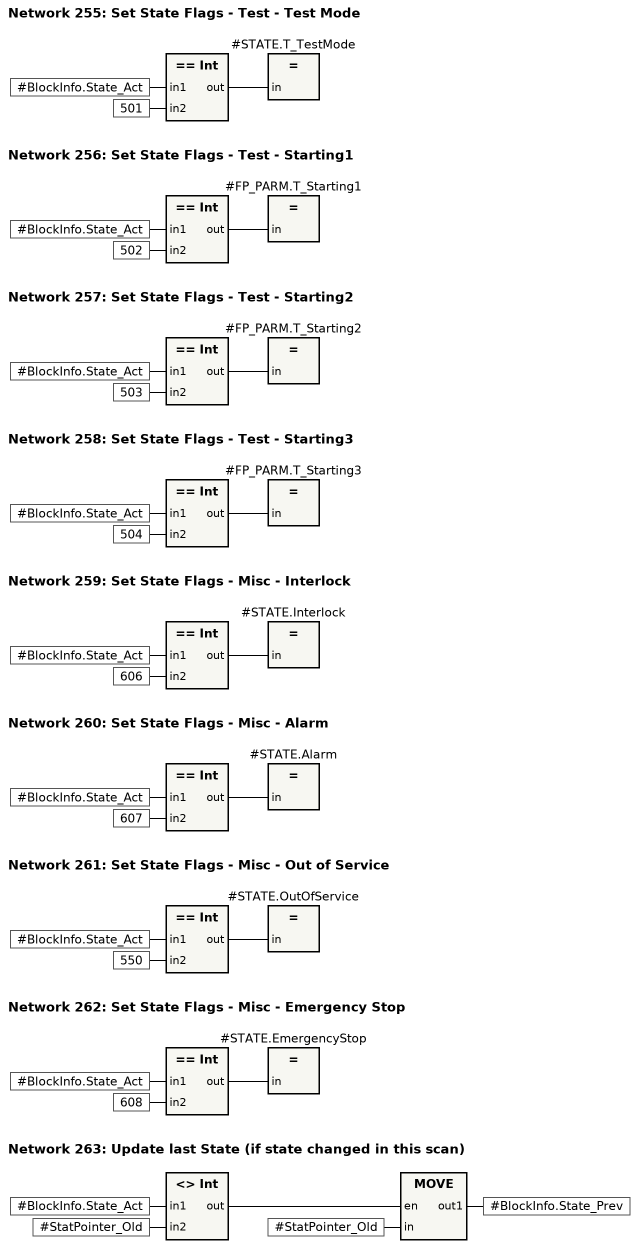
   #STATE.T_TestMode := #BlockInfo.State_Act = 501;
END_REGION

REGION Network 256: Set State Flags - Test - Starting1
   #FP_PARM.T_Starting1 := #BlockInfo.State_Act = 502;
END_REGION

REGION Network 257: Set State Flags - Test - Starting2
   #FP_PARM.T_Starting2 := #BlockInfo.State_Act = 503;
END_REGION

REGION Network 258: Set State Flags - Test - Starting3
   #FP_PARM.T_Starting3 := #BlockInfo.State_Act = 504;
END_REGION

REGION Network 259: Set State Flags - Misc - Interlock
   #STATE.Interlock := #BlockInfo.State_Act = 606;
END_REGION

REGION Network 260: Set State Flags - Misc - Alarm
   #STATE.Alarm := #BlockInfo.State_Act = 607;
END_REGION

REGION Network 261: Set State Flags - Misc - Out of Service
   #STATE.OutOfService := #BlockInfo.State_Act = 550;
END_REGION

REGION Network 262: Set State Flags - Misc - Emergency Stop
   #STATE.EmergencyStop := #BlockInfo.State_Act = 608;
END_REGION

REGION Network 263: Update last State (if state changed in this scan)
   IF #BlockInfo.State_Act <> #StatPointer_Old THEN #BlockInfo.State_Prev := #StatPointer_Old; END_IF;
END_REGION

REGION Network 264: Update MSW
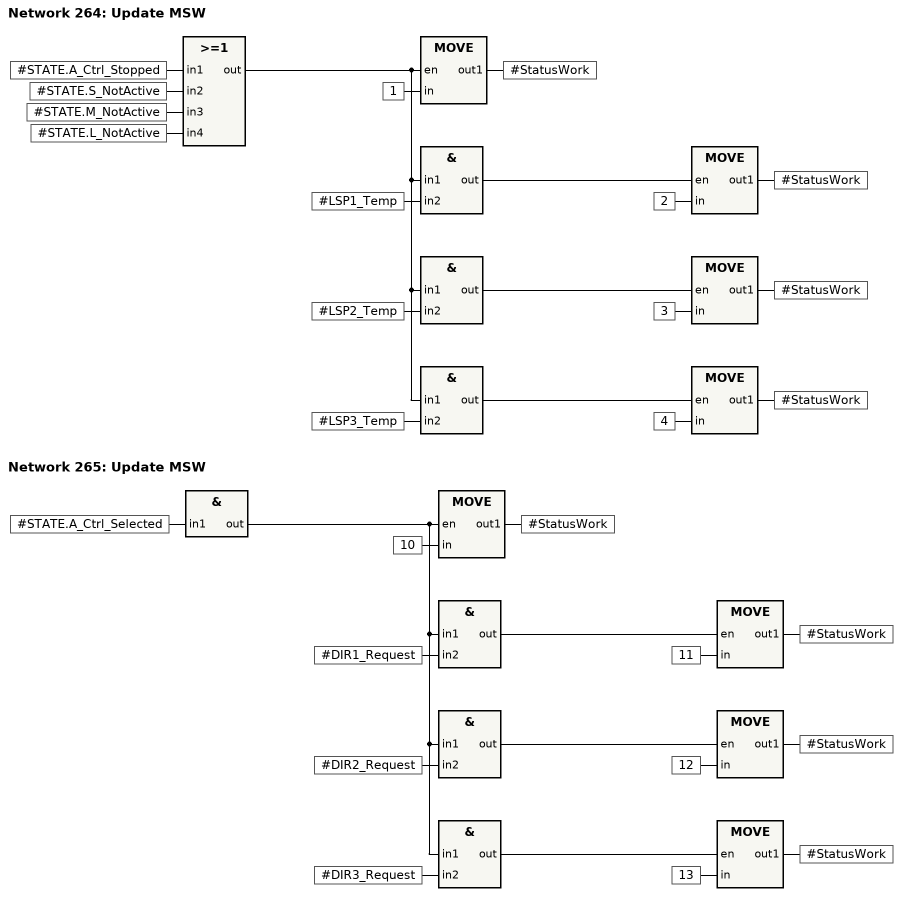
   #_w1 := #STATE.A_Ctrl_Stopped OR #STATE.S_NotActive OR #STATE.M_NotActive OR #STATE.L_NotActive;
   IF #_w1 THEN #StatusWork := 1; END_IF;
   IF #_w1 AND #LSP1_Temp THEN #StatusWork := 2; END_IF;
   IF #_w1 AND #LSP2_Temp THEN #StatusWork := 3; END_IF;
   IF #_w1 AND #LSP3_Temp THEN #StatusWork := 4; END_IF;
END_REGION

REGION Network 265: Update MSW
   IF #STATE.A_Ctrl_Selected THEN #StatusWork := 10; END_IF;
   IF #STATE.A_Ctrl_Selected AND #DIR1_Request THEN #StatusWork := 11; END_IF;
   IF #STATE.A_Ctrl_Selected AND #DIR2_Request THEN #StatusWork := 12; END_IF;
   IF #STATE.A_Ctrl_Selected AND #DIR3_Request THEN #StatusWork := 13; END_IF;
END_REGION

REGION Network 266: Update MSW
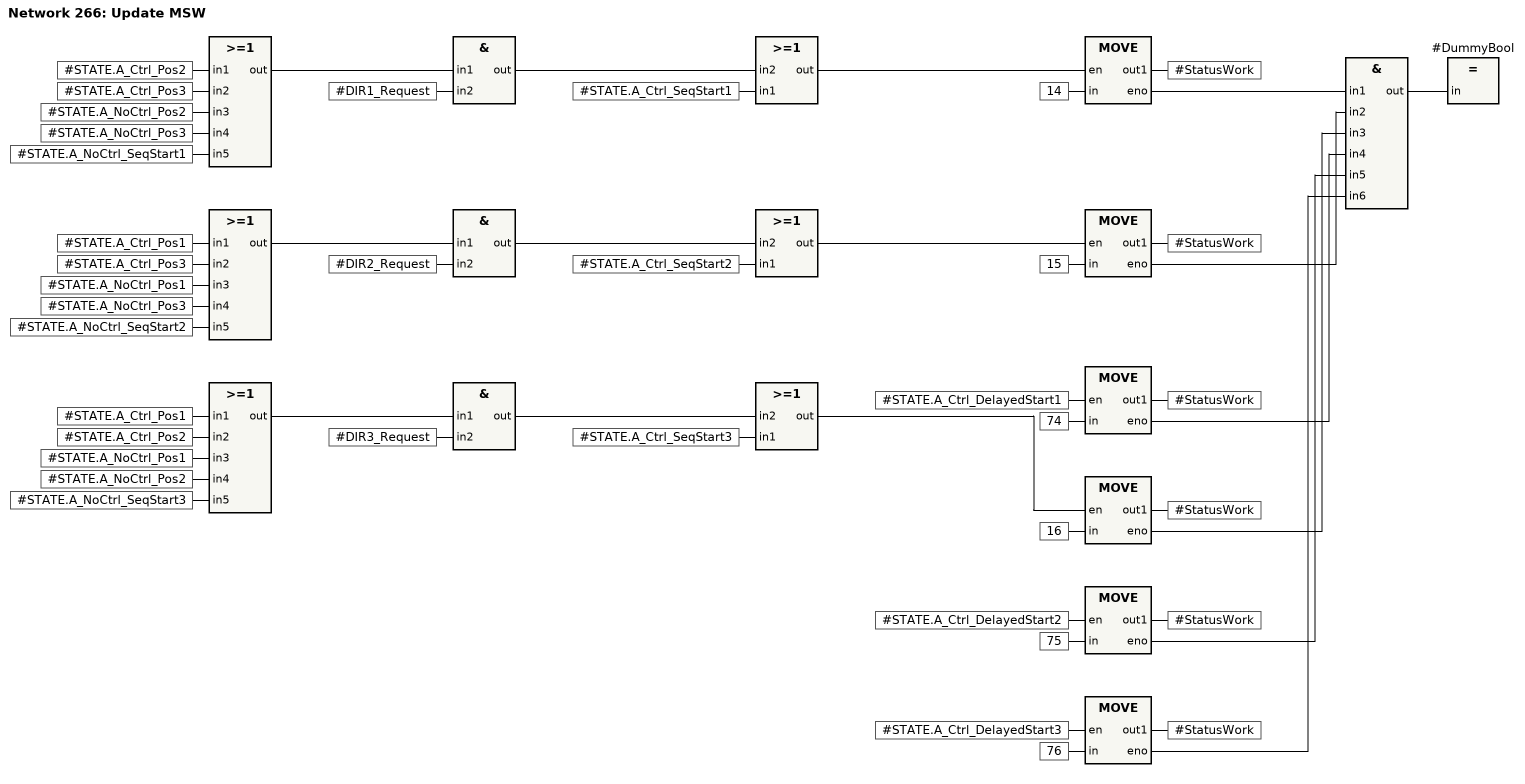
   // ENO of a box is taken as its EN; it also drops when the box reports an error
   #_w1 := ((#STATE.A_Ctrl_Pos2 OR #STATE.A_Ctrl_Pos3 OR #STATE.A_NoCtrl_Pos2 OR #STATE.A_NoCtrl_Pos3 OR #STATE.A_NoCtrl_SeqStart1) AND #DIR1_Request) OR #STATE.A_Ctrl_SeqStart1;
   IF #_w1 THEN #StatusWork := 14; END_IF;
   #_w2 := ((#STATE.A_Ctrl_Pos1 OR #STATE.A_Ctrl_Pos3 OR #STATE.A_NoCtrl_Pos1 OR #STATE.A_NoCtrl_Pos3 OR #STATE.A_NoCtrl_SeqStart2) AND #DIR2_Request) OR #STATE.A_Ctrl_SeqStart2;
   IF #_w2 THEN #StatusWork := 15; END_IF;
   #_w3 := ((#STATE.A_Ctrl_Pos1 OR #STATE.A_Ctrl_Pos2 OR #STATE.A_NoCtrl_Pos1 OR #STATE.A_NoCtrl_Pos2 OR #STATE.A_NoCtrl_SeqStart3) AND #DIR3_Request) OR #STATE.A_Ctrl_SeqStart3;
   IF #_w3 THEN #StatusWork := 16; END_IF;
   IF #STATE.A_Ctrl_DelayedStart1 THEN #StatusWork := 74; END_IF;
   IF #STATE.A_Ctrl_DelayedStart2 THEN #StatusWork := 75; END_IF;
   IF #STATE.A_Ctrl_DelayedStart3 THEN #StatusWork := 76; END_IF;
   #DummyBool := #_w1 AND #_w2 AND #_w3 AND #STATE.A_Ctrl_DelayedStart1 AND #STATE.A_Ctrl_DelayedStart2 AND #STATE.A_Ctrl_DelayedStart3;
END_REGION

REGION Network 267: Update MSW
   // Build 007 - 30.09.2020 (EXTBOB):  State Alarm Neg added to avoid start warn in case of alarm state
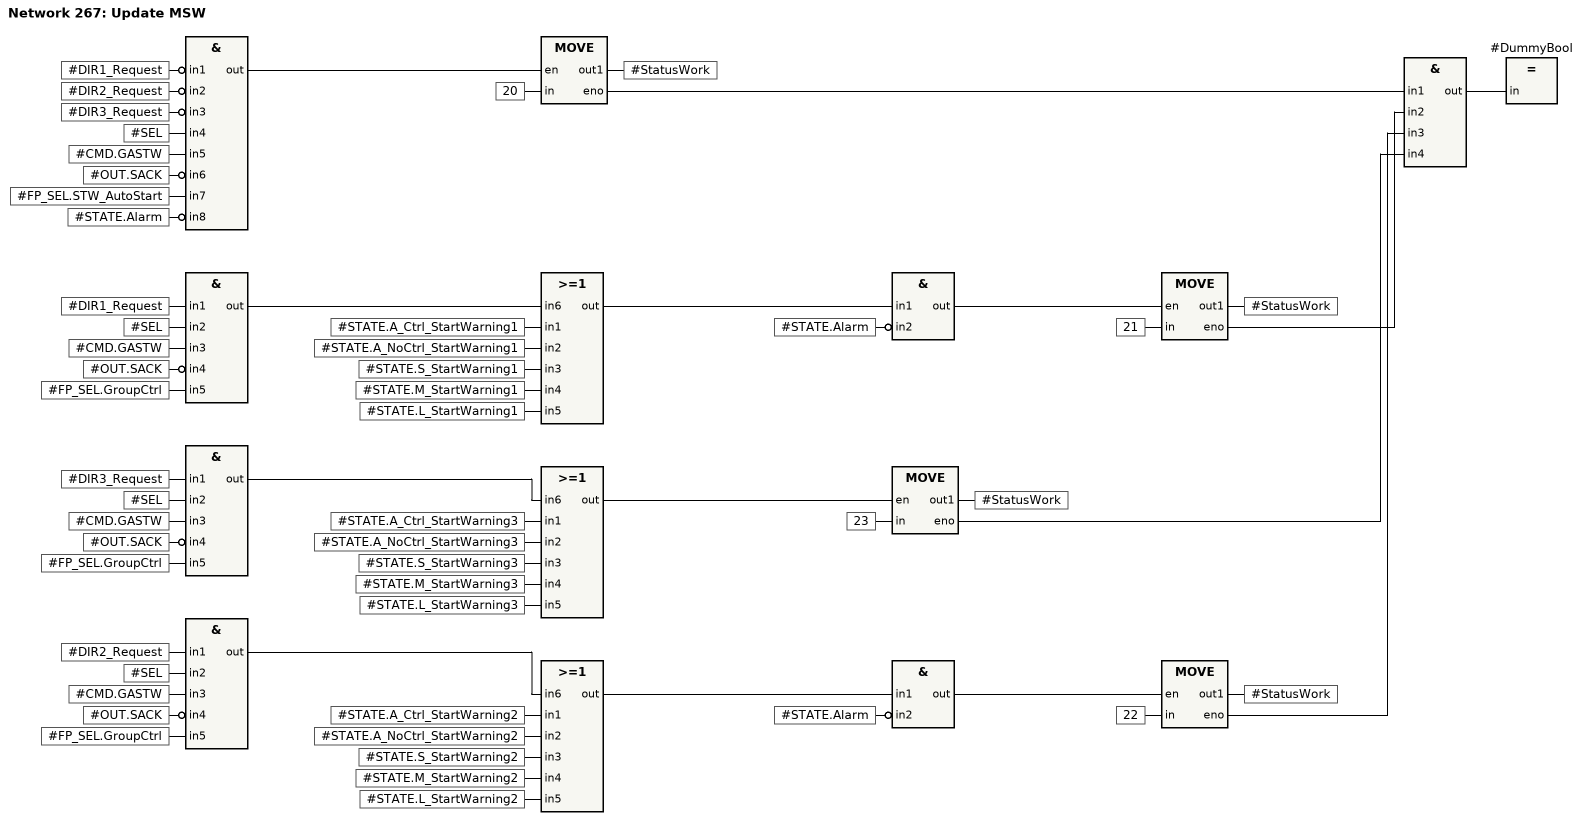
   // ENO of a box is taken as its EN; it also drops when the box reports an error
   #_w1 := NOT #DIR1_Request AND NOT #DIR2_Request AND NOT #DIR3_Request AND #SEL AND #CMD.GASTW AND NOT #OUT.SACK AND #FP_SEL.STW_AutoStart AND NOT #STATE.Alarm;
   IF #_w1 THEN #StatusWork := 20; END_IF;
   #_w2 := ((#DIR1_Request AND #SEL AND #CMD.GASTW AND NOT #OUT.SACK AND #FP_SEL.GroupCtrl) OR #STATE.A_Ctrl_StartWarning1 OR #STATE.A_NoCtrl_StartWarning1 OR #STATE.S_StartWarning1 OR #STATE.M_StartWarning1 OR #STATE.L_StartWarning1) AND NOT #STATE.Alarm;
   IF #_w2 THEN #StatusWork := 21; END_IF;
   #_w3 := ((#DIR2_Request AND #SEL AND #CMD.GASTW AND NOT #OUT.SACK AND #FP_SEL.GroupCtrl) OR #STATE.A_Ctrl_StartWarning2 OR #STATE.A_NoCtrl_StartWarning2 OR #STATE.S_StartWarning2 OR #STATE.M_StartWarning2 OR #STATE.L_StartWarning2) AND NOT #STATE.Alarm;
   IF #_w3 THEN #StatusWork := 22; END_IF;
   #_w4 := (#DIR3_Request AND #SEL AND #CMD.GASTW AND NOT #OUT.SACK AND #FP_SEL.GroupCtrl) OR #STATE.A_Ctrl_StartWarning3 OR #STATE.A_NoCtrl_StartWarning3 OR #STATE.S_StartWarning3 OR #STATE.M_StartWarning3 OR #STATE.L_StartWarning3;
   IF #_w4 THEN #StatusWork := 23; END_IF;
   #DummyBool := #_w1 AND #_w2 AND #_w3 AND #_w4;
END_REGION

REGION Network 268: Update MSW
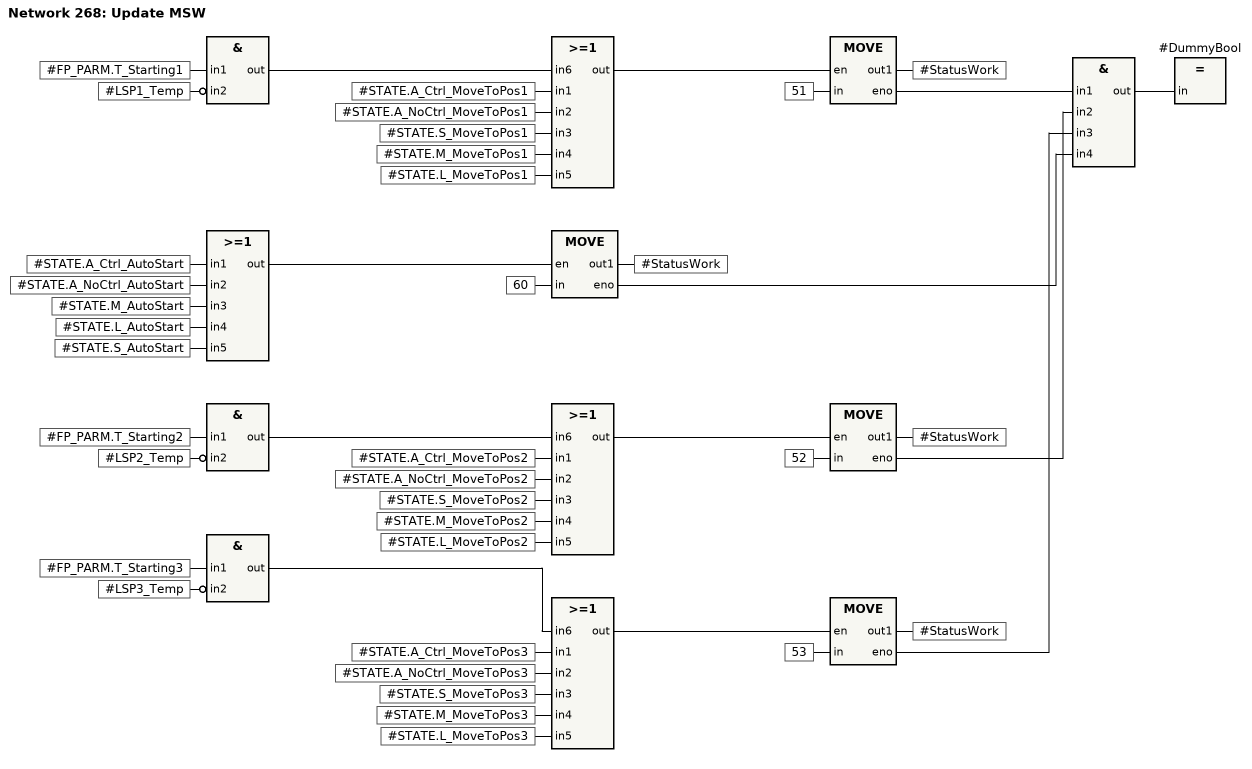
   // ENO of a box is taken as its EN; it also drops when the box reports an error
   #_w1 := (#FP_PARM.T_Starting1 AND NOT #LSP1_Temp) OR #STATE.A_Ctrl_MoveToPos1 OR #STATE.A_NoCtrl_MoveToPos1 OR #STATE.S_MoveToPos1 OR #STATE.M_MoveToPos1 OR #STATE.L_MoveToPos1;
   IF #_w1 THEN #StatusWork := 51; END_IF;
   #_w2 := (#FP_PARM.T_Starting2 AND NOT #LSP2_Temp) OR #STATE.A_Ctrl_MoveToPos2 OR #STATE.A_NoCtrl_MoveToPos2 OR #STATE.S_MoveToPos2 OR #STATE.M_MoveToPos2 OR #STATE.L_MoveToPos2;
   IF #_w2 THEN #StatusWork := 52; END_IF;
   #_w3 := (#FP_PARM.T_Starting3 AND NOT #LSP3_Temp) OR #STATE.A_Ctrl_MoveToPos3 OR #STATE.A_NoCtrl_MoveToPos3 OR #STATE.S_MoveToPos3 OR #STATE.M_MoveToPos3 OR #STATE.L_MoveToPos3;
   IF #_w3 THEN #StatusWork := 53; END_IF;
   #_w4 := #STATE.A_Ctrl_AutoStart OR #STATE.A_NoCtrl_AutoStart OR #STATE.M_AutoStart OR #STATE.L_AutoStart OR #STATE.S_AutoStart;
   IF #_w4 THEN #StatusWork := 60; END_IF;
   #DummyBool := #_w1 AND #_w2 AND #_w3 AND #_w4;
END_REGION

REGION Network 269: Update MSW
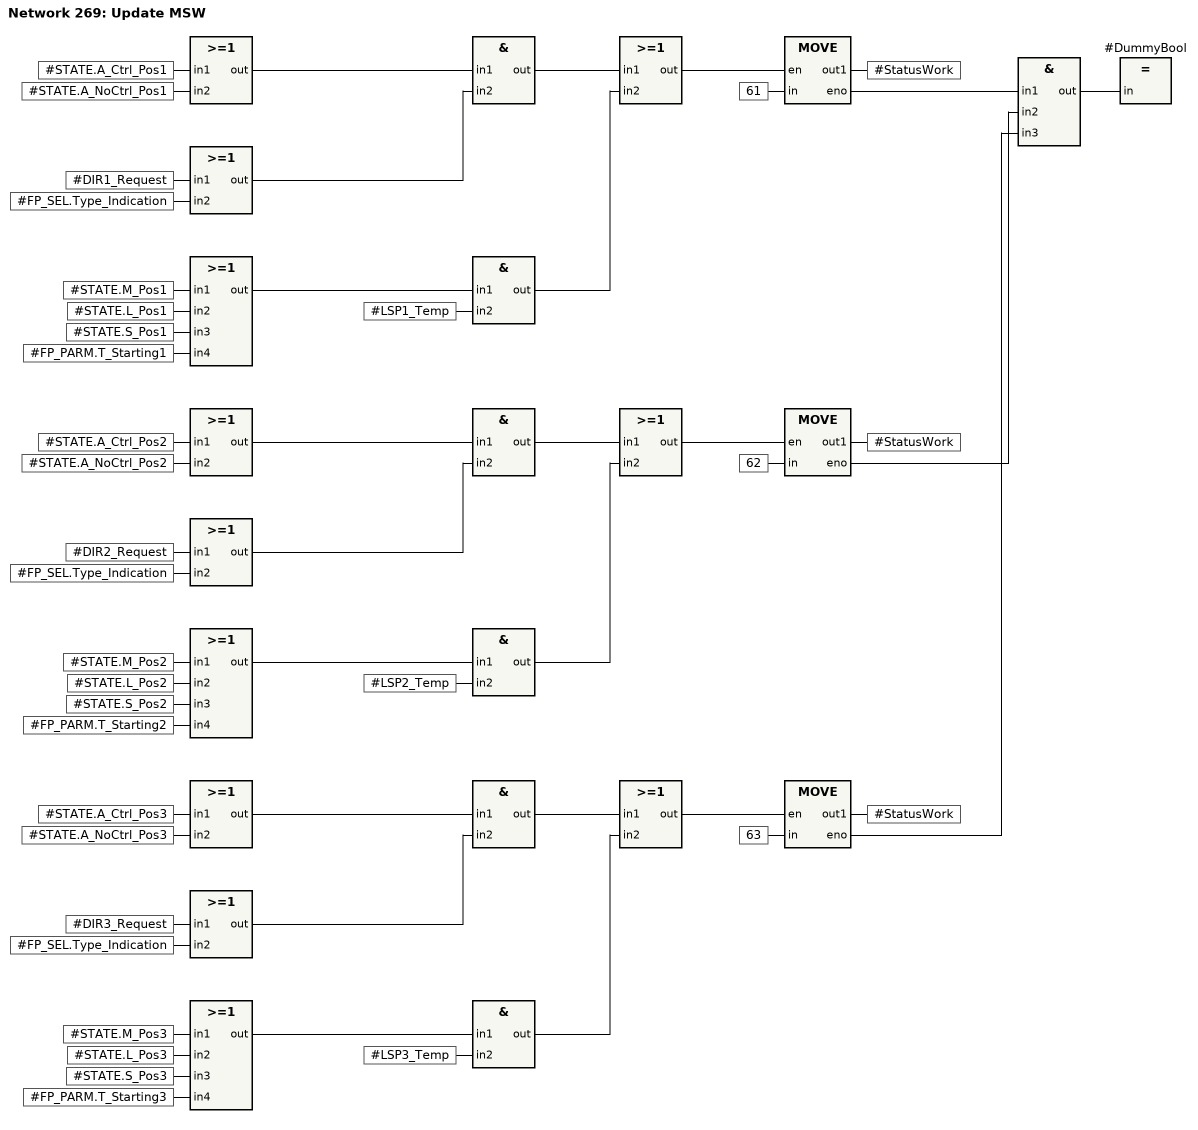
   // ENO of a box is taken as its EN; it also drops when the box reports an error
   #_w1 := ((#STATE.A_Ctrl_Pos1 OR #STATE.A_NoCtrl_Pos1) AND (#DIR1_Request OR #FP_SEL.Type_Indication)) OR ((#STATE.M_Pos1 OR #STATE.L_Pos1 OR #STATE.S_Pos1 OR #FP_PARM.T_Starting1) AND #LSP1_Temp);
   IF #_w1 THEN #StatusWork := 61; END_IF;
   #_w2 := ((#STATE.A_Ctrl_Pos2 OR #STATE.A_NoCtrl_Pos2) AND (#DIR2_Request OR #FP_SEL.Type_Indication)) OR ((#STATE.M_Pos2 OR #STATE.L_Pos2 OR #STATE.S_Pos2 OR #FP_PARM.T_Starting2) AND #LSP2_Temp);
   IF #_w2 THEN #StatusWork := 62; END_IF;
   #_w3 := ((#STATE.A_Ctrl_Pos3 OR #STATE.A_NoCtrl_Pos3) AND (#DIR3_Request OR #FP_SEL.Type_Indication)) OR ((#STATE.M_Pos3 OR #STATE.L_Pos3 OR #STATE.S_Pos3 OR #FP_PARM.T_Starting3) AND #LSP3_Temp);
   IF #_w3 THEN #StatusWork := 63; END_IF;
   #DummyBool := #_w1 AND #_w2 AND #_w3;
END_REGION

REGION Network 270: Update MSW
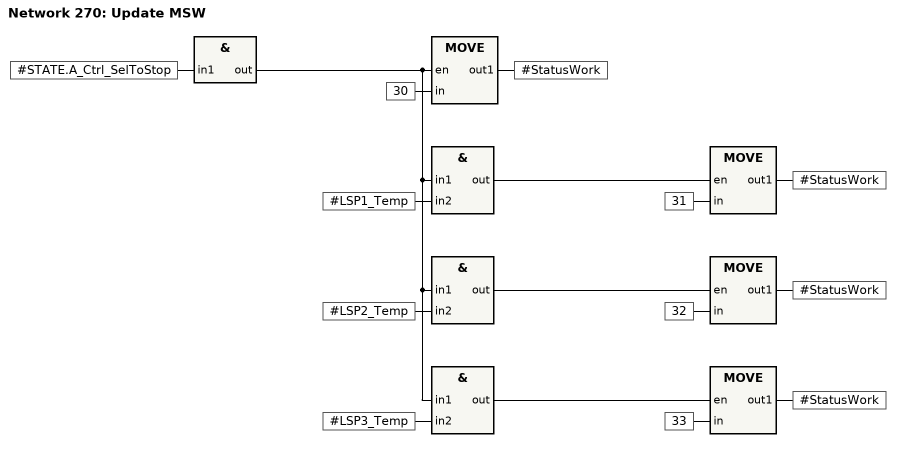
   IF #STATE.A_Ctrl_SelToStop THEN #StatusWork := 30; END_IF;
   IF #STATE.A_Ctrl_SelToStop AND #LSP1_Temp THEN #StatusWork := 31; END_IF;
   IF #STATE.A_Ctrl_SelToStop AND #LSP2_Temp THEN #StatusWork := 32; END_IF;
   IF #STATE.A_Ctrl_SelToStop AND #LSP3_Temp THEN #StatusWork := 33; END_IF;
END_REGION

REGION Network 271: Update MSW
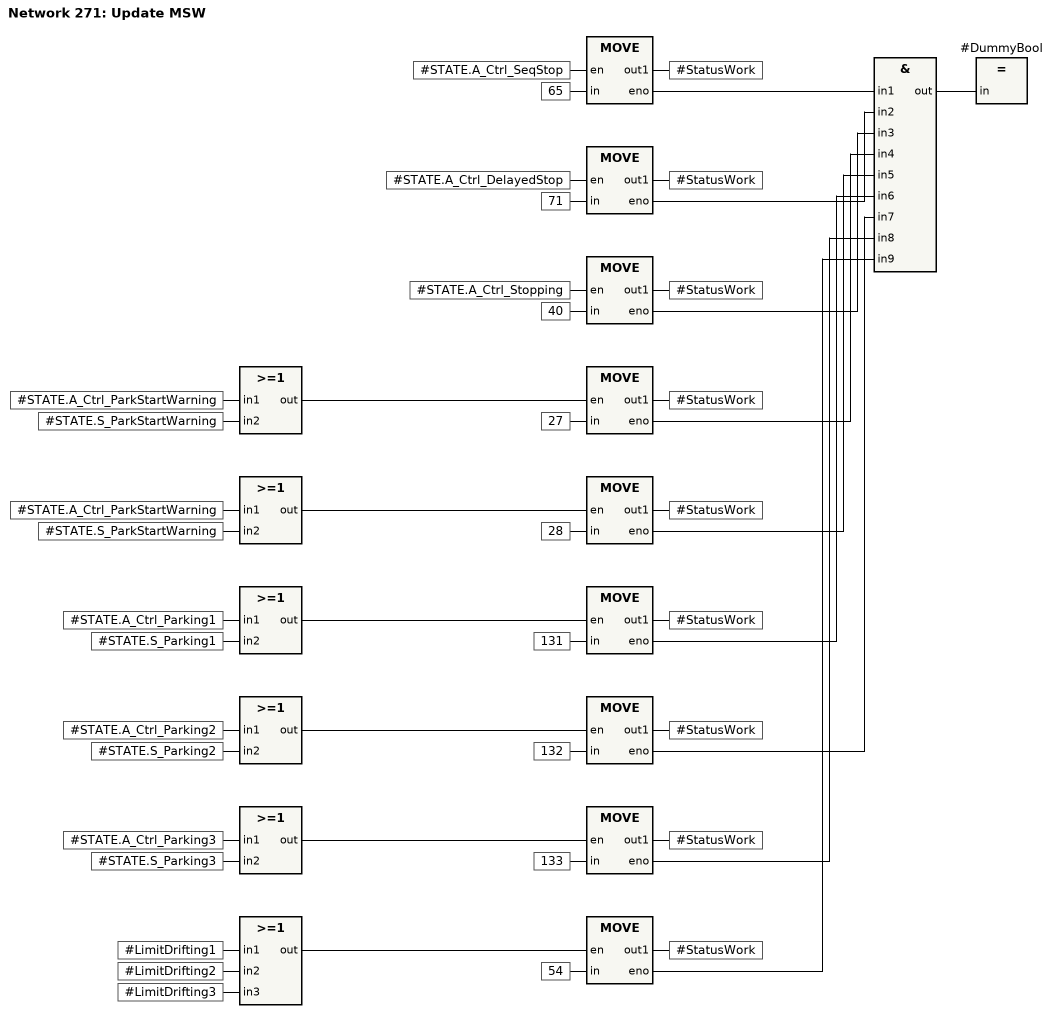
   // ENO of a box is taken as its EN; it also drops when the box reports an error
   IF #STATE.A_Ctrl_SeqStop THEN #StatusWork := 65; END_IF;
   IF #STATE.A_Ctrl_DelayedStop THEN #StatusWork := 71; END_IF;
   IF #STATE.A_Ctrl_Stopping THEN #StatusWork := 40; END_IF;
   #_w1 := #STATE.A_Ctrl_ParkStartWarning OR #STATE.S_ParkStartWarning;
   IF #_w1 THEN #StatusWork := 27; END_IF;
   #_w2 := #STATE.A_Ctrl_ParkStartWarning OR #STATE.S_ParkStartWarning;
   IF #_w2 THEN #StatusWork := 28; END_IF;
   #_w3 := #STATE.A_Ctrl_Parking1 OR #STATE.S_Parking1;
   IF #_w3 THEN #StatusWork := 131; END_IF;
   #_w4 := #STATE.A_Ctrl_Parking2 OR #STATE.S_Parking2;
   IF #_w4 THEN #StatusWork := 132; END_IF;
   #_w5 := #STATE.A_Ctrl_Parking3 OR #STATE.S_Parking3;
   IF #_w5 THEN #StatusWork := 133; END_IF;
   #_w6 := #LimitDrifting1 OR #LimitDrifting2 OR #LimitDrifting3;
   IF #_w6 THEN #StatusWork := 54; END_IF;
   #DummyBool := #STATE.A_Ctrl_SeqStop AND #STATE.A_Ctrl_DelayedStop AND #STATE.A_Ctrl_Stopping AND #_w1 AND #_w2 AND #_w3 AND #_w4 AND #_w5 AND #_w6;
END_REGION

REGION Network 272: Update MSW
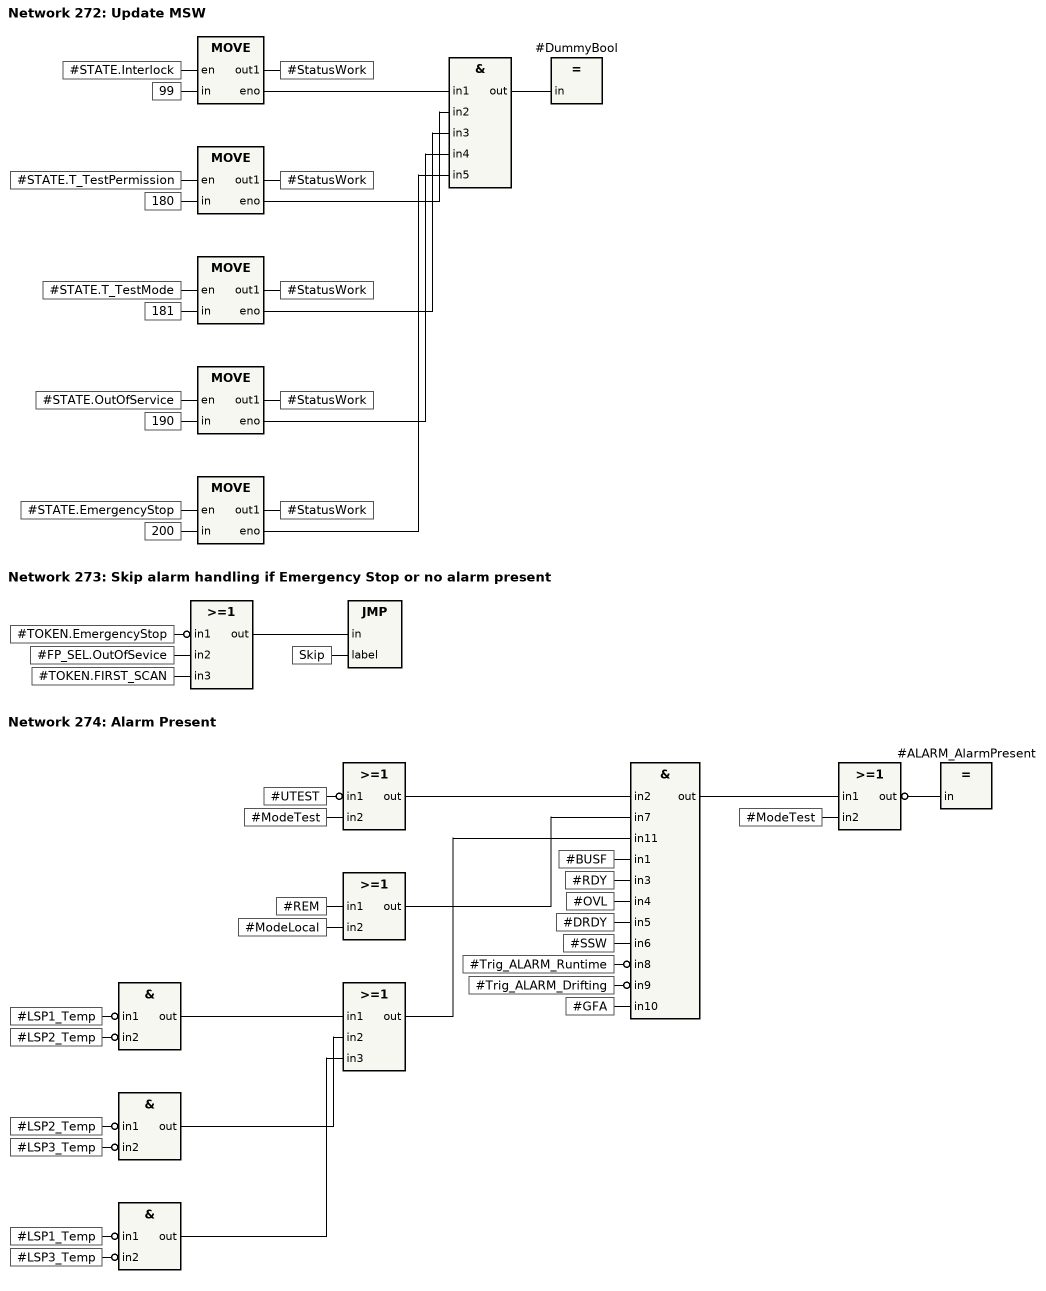
   // ENO of a box is taken as its EN; it also drops when the box reports an error
   IF #STATE.Interlock THEN #StatusWork := 99; END_IF;
   IF #STATE.T_TestPermission THEN #StatusWork := 180; END_IF;
   IF #STATE.T_TestMode THEN #StatusWork := 181; END_IF;
   IF #STATE.OutOfService THEN #StatusWork := 190; END_IF;
   IF #STATE.EmergencyStop THEN #StatusWork := 200; END_IF;
   #DummyBool := #STATE.Interlock AND #STATE.T_TestPermission AND #STATE.T_TestMode AND #STATE.OutOfService AND #STATE.EmergencyStop;
END_REGION

REGION Network 273: Skip alarm handling if Emergency Stop or no alarm present
   // Skip = Skip Alarm
   IF NOT #TOKEN.EmergencyStop OR #FP_SEL.OutOfSevice OR #TOKEN.FIRST_SCAN THEN GOTO Skip; END_IF;
END_REGION

REGION Network 274: Alarm Present
   #ALARM_AlarmPresent := NOT (((NOT #UTEST OR #ModeTest) AND (#REM OR #ModeLocal) AND ((NOT #LSP1_Temp AND NOT #LSP2_Temp) OR (NOT #LSP2_Temp AND NOT #LSP3_Temp) OR (NOT #LSP1_Temp AND NOT #LSP3_Temp)) AND #BUSF AND #RDY AND #OVL AND #DRDY AND #SSW AND NOT #Trig_ALARM_Runtime AND NOT #Trig_ALARM_Drifting AND #GFA) OR #ModeTest);
END_REGION

REGION Network 275: Alarm Warn Present
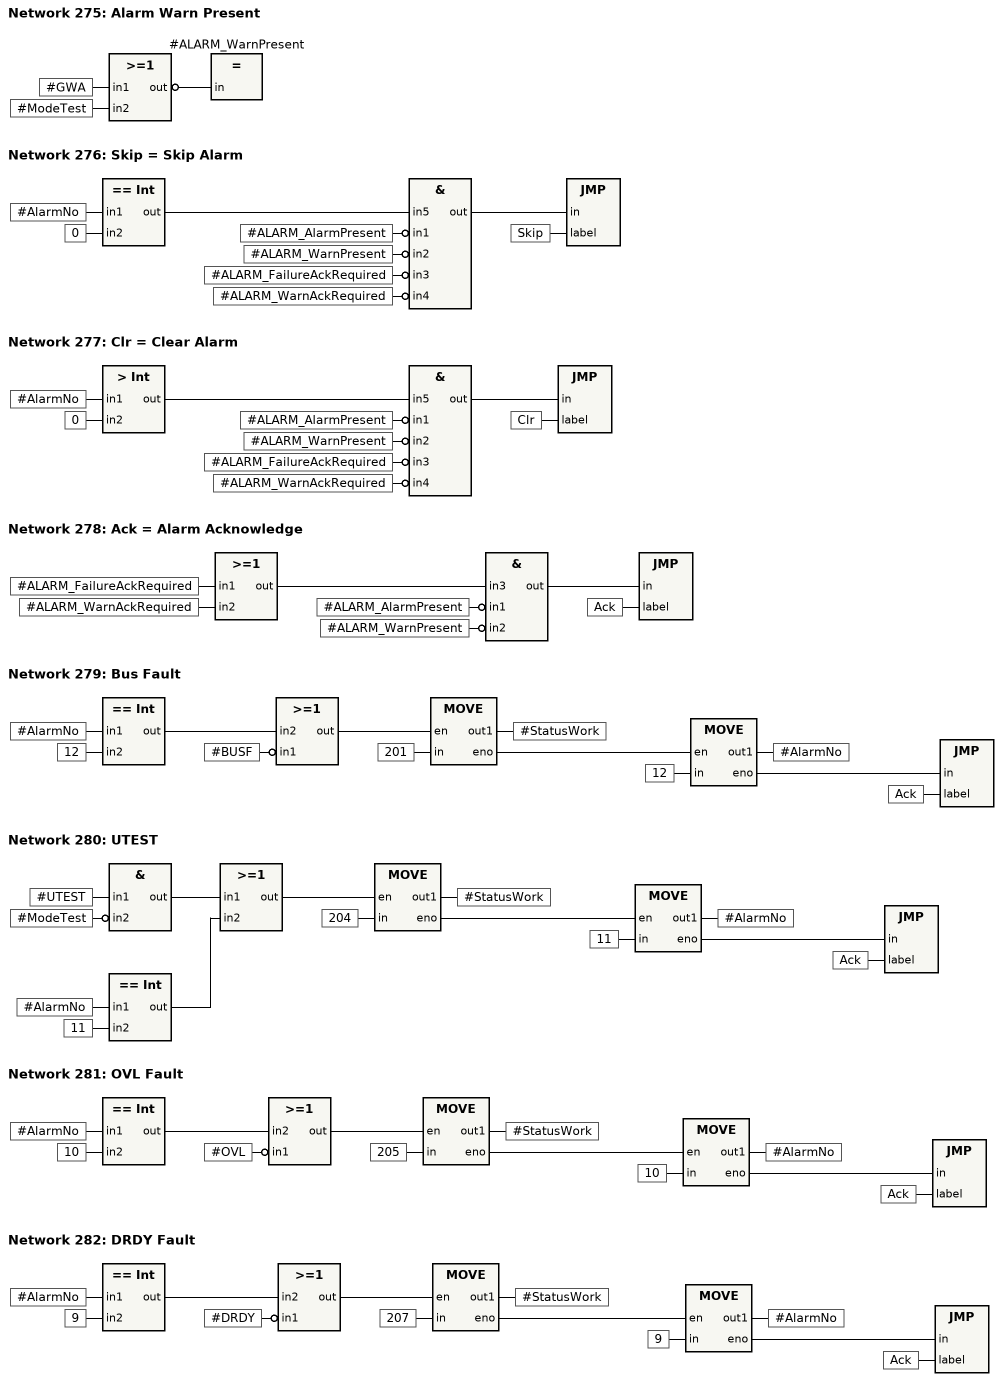
   #ALARM_WarnPresent := NOT (#GWA OR #ModeTest);
END_REGION

REGION Network 276: Skip = Skip Alarm
   IF (#AlarmNo = 0) AND NOT #ALARM_AlarmPresent AND NOT #ALARM_WarnPresent AND NOT #ALARM_FailureAckRequired AND NOT #ALARM_WarnAckRequired THEN
       GOTO Skip;
   END_IF;
END_REGION

REGION Network 277: Clr = Clear Alarm
   IF (#AlarmNo > 0) AND NOT #ALARM_AlarmPresent AND NOT #ALARM_WarnPresent AND NOT #ALARM_FailureAckRequired AND NOT #ALARM_WarnAckRequired THEN
       GOTO Clr;
   END_IF;
END_REGION

REGION Network 278: Ack = Alarm Acknowledge
   IF (#ALARM_FailureAckRequired OR #ALARM_WarnAckRequired) AND NOT #ALARM_AlarmPresent AND NOT #ALARM_WarnPresent THEN
       GOTO Ack;
   END_IF;
END_REGION

REGION Network 279: Bus Fault
   // ENO of a box is taken as its EN; it also drops when the box reports an error
   #_w1 := (#AlarmNo = 12) OR NOT #BUSF;
   IF #_w1 THEN
       #StatusWork := 201;
       #AlarmNo := 12;
       GOTO Ack;
   END_IF;
END_REGION

REGION Network 280: UTEST
   // ENO of a box is taken as its EN; it also drops when the box reports an error
   #_w1 := (#UTEST AND NOT #ModeTest) OR (#AlarmNo = 11);
   IF #_w1 THEN
       #StatusWork := 204;
       #AlarmNo := 11;
       GOTO Ack;
   END_IF;
END_REGION

REGION Network 281: OVL Fault
   // ENO of a box is taken as its EN; it also drops when the box reports an error
   #_w1 := (#AlarmNo = 10) OR NOT #OVL;
   IF #_w1 THEN
       #StatusWork := 205;
       #AlarmNo := 10;
       GOTO Ack;
   END_IF;
END_REGION

REGION Network 282: DRDY Fault
   // ENO of a box is taken as its EN; it also drops when the box reports an error
   #_w1 := (#AlarmNo = 9) OR NOT #DRDY;
   IF #_w1 THEN
       #StatusWork := 207;
       #AlarmNo := 9;
       GOTO Ack;
   END_IF;
END_REGION

REGION Network 283: RDY Fault
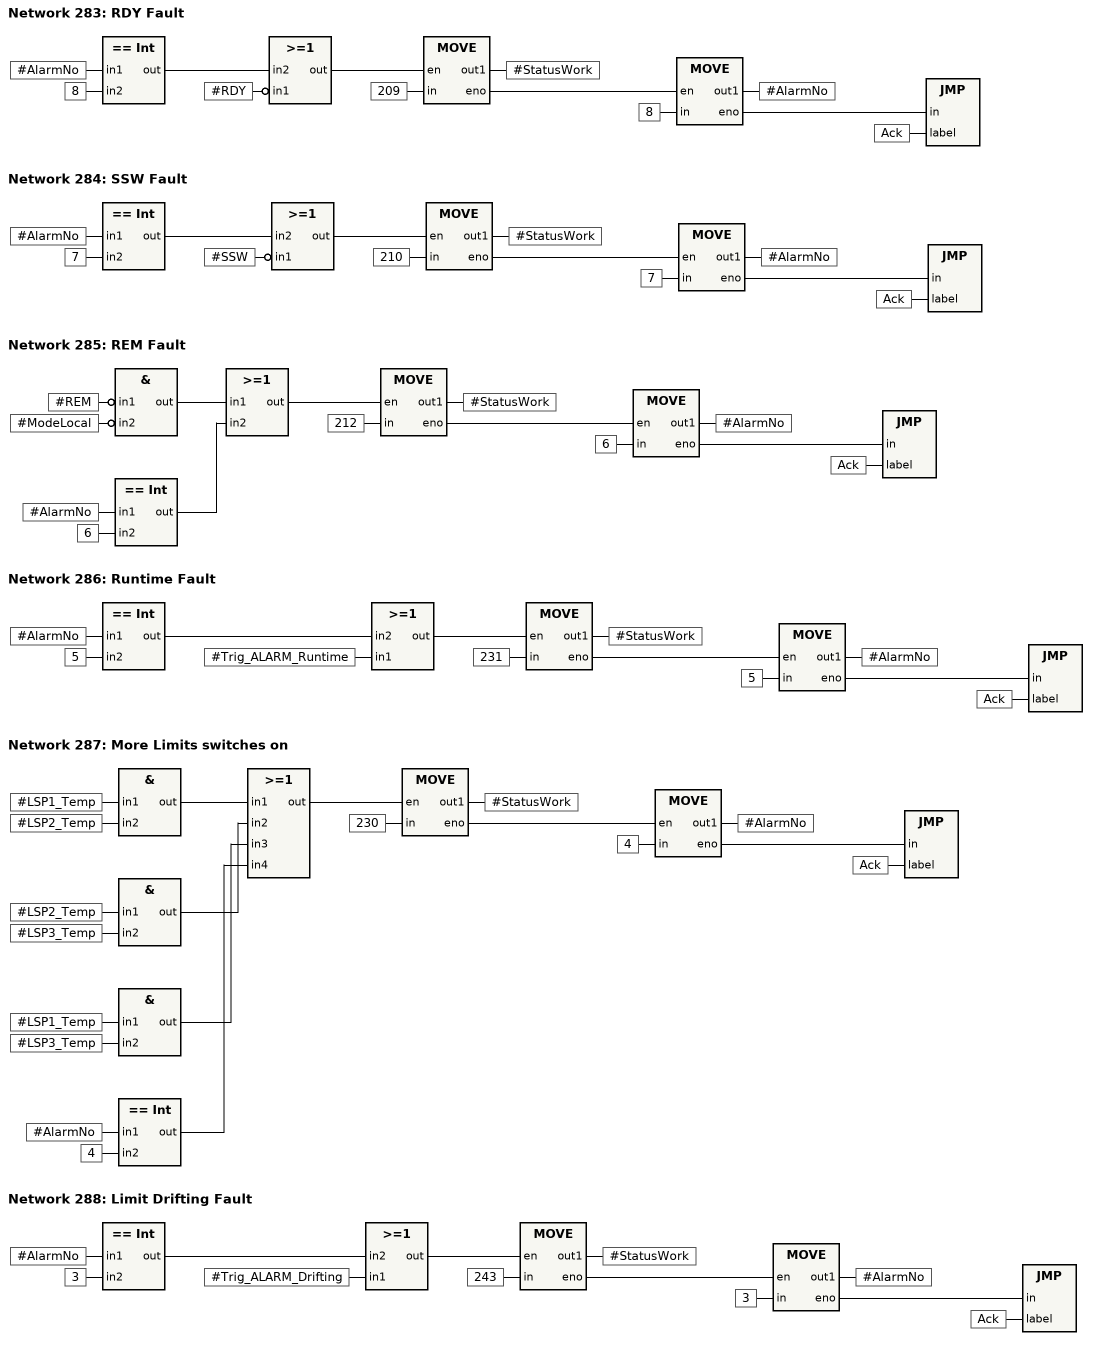
   // ENO of a box is taken as its EN; it also drops when the box reports an error
   #_w1 := (#AlarmNo = 8) OR NOT #RDY;
   IF #_w1 THEN
       #StatusWork := 209;
       #AlarmNo := 8;
       GOTO Ack;
   END_IF;
END_REGION

REGION Network 284: SSW Fault
   // ENO of a box is taken as its EN; it also drops when the box reports an error
   #_w1 := (#AlarmNo = 7) OR NOT #SSW;
   IF #_w1 THEN
       #StatusWork := 210;
       #AlarmNo := 7;
       GOTO Ack;
   END_IF;
END_REGION

REGION Network 285: REM Fault
   // ENO of a box is taken as its EN; it also drops when the box reports an error
   #_w1 := (NOT #REM AND NOT #ModeLocal) OR (#AlarmNo = 6);
   IF #_w1 THEN
       #StatusWork := 212;
       #AlarmNo := 6;
       GOTO Ack;
   END_IF;
END_REGION

REGION Network 286: Runtime Fault
   // ENO of a box is taken as its EN; it also drops when the box reports an error
   #_w1 := (#AlarmNo = 5) OR #Trig_ALARM_Runtime;
   IF #_w1 THEN
       #StatusWork := 231;
       #AlarmNo := 5;
       GOTO Ack;
   END_IF;
END_REGION

REGION Network 287: More Limits switches on
   // ENO of a box is taken as its EN; it also drops when the box reports an error
   #_w1 := (#LSP1_Temp AND #LSP2_Temp) OR (#LSP2_Temp AND #LSP3_Temp) OR (#LSP1_Temp AND #LSP3_Temp) OR (#AlarmNo = 4);
   IF #_w1 THEN
       #StatusWork := 230;
       #AlarmNo := 4;
       GOTO Ack;
   END_IF;
END_REGION

REGION Network 288: Limit Drifting Fault
   // ENO of a box is taken as its EN; it also drops when the box reports an error
   #_w1 := (#AlarmNo = 3) OR #Trig_ALARM_Drifting;
   IF #_w1 THEN
       #StatusWork := 243;
       #AlarmNo := 3;
       GOTO Ack;
   END_IF;
END_REGION

REGION Network 289: GFA Fault
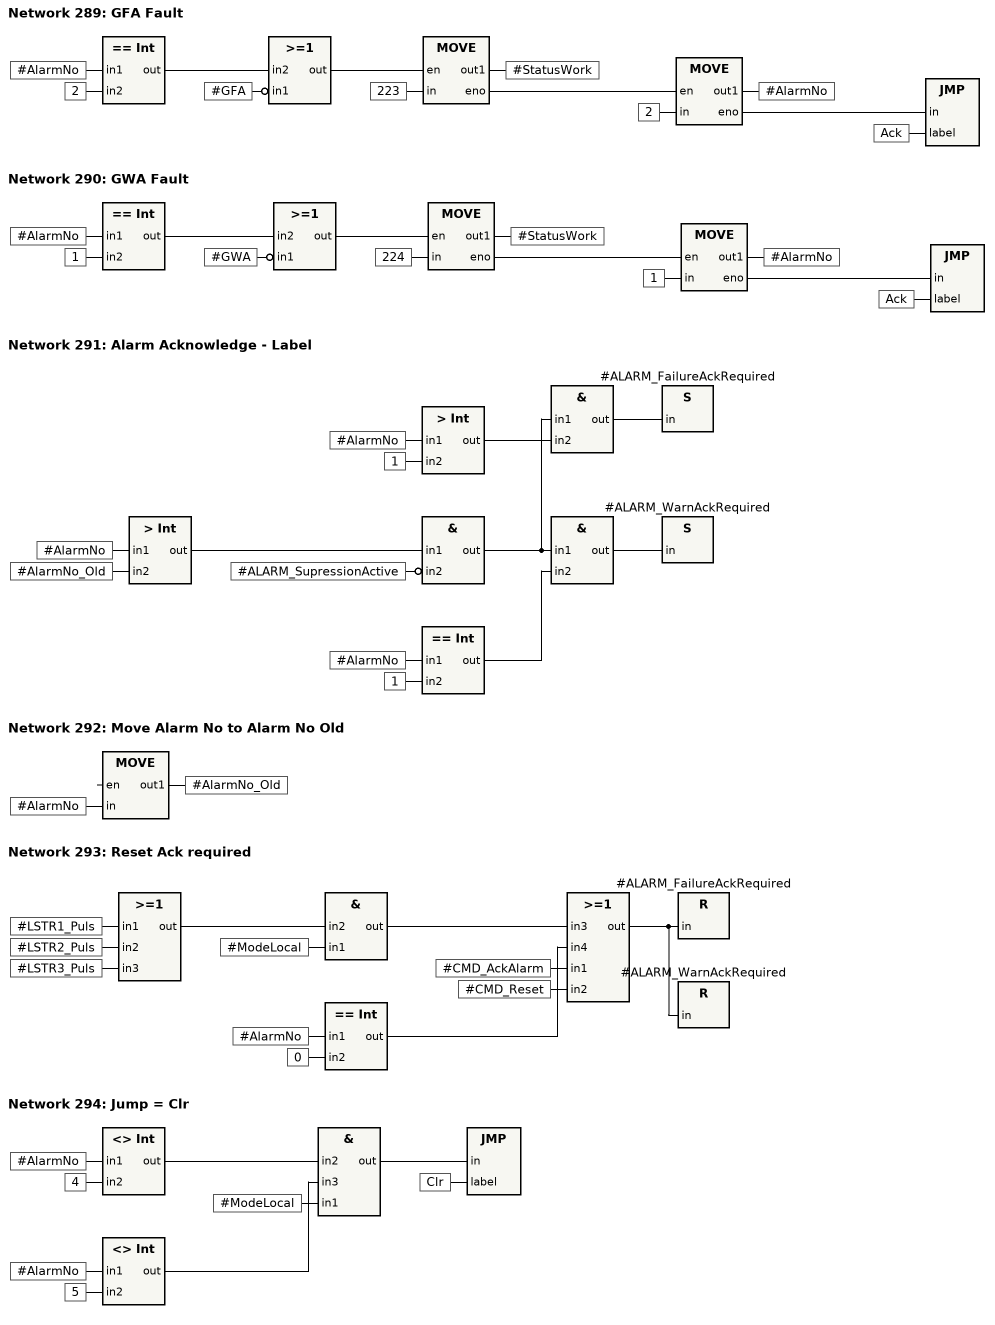
   // ENO of a box is taken as its EN; it also drops when the box reports an error
   #_w1 := (#AlarmNo = 2) OR NOT #GFA;
   IF #_w1 THEN
       #StatusWork := 223;
       #AlarmNo := 2;
       GOTO Ack;
   END_IF;
END_REGION

REGION Network 290: GWA Fault
   // ENO of a box is taken as its EN; it also drops when the box reports an error
   #_w1 := (#AlarmNo = 1) OR NOT #GWA;
   IF #_w1 THEN
       #StatusWork := 224;
       #AlarmNo := 1;
       GOTO Ack;
   END_IF;
END_REGION

REGION Network 291: Alarm Acknowledge - Label
   Ack:
   #_w1 := (#AlarmNo > #AlarmNo_Old) AND NOT #ALARM_SupressionActive;
   IF #_w1 AND (#AlarmNo > 1) THEN #ALARM_FailureAckRequired := TRUE; END_IF;
   IF #_w1 AND (#AlarmNo = 1) THEN #ALARM_WarnAckRequired := TRUE; END_IF;
END_REGION

REGION Network 292: Move Alarm No to Alarm No Old
   #AlarmNo_Old := #AlarmNo;
END_REGION

REGION Network 293: Reset Ack required
   IF ((#LSTR1_Puls OR #LSTR2_Puls OR #LSTR3_Puls) AND #ModeLocal) OR (#AlarmNo = 0) OR #CMD_AckAlarm OR #CMD_Reset THEN
       #ALARM_FailureAckRequired := FALSE;
       #ALARM_WarnAckRequired := FALSE;
   END_IF;
END_REGION

REGION Network 294: Jump = Clr
   IF (#AlarmNo <> 4) AND (#AlarmNo <> 5) AND #ModeLocal THEN GOTO Clr; END_IF;
END_REGION

REGION Network 295: Skip = Skip Alarm
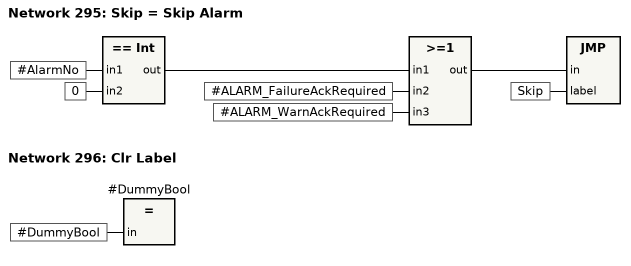
   IF (#AlarmNo = 0) OR #ALARM_FailureAckRequired OR #ALARM_WarnAckRequired THEN GOTO Skip; END_IF;
END_REGION

REGION Network 296: Clr Label
   Clr:
   #DummyBool := #DummyBool;
END_REGION

REGION Network 297: Clear Alarm No
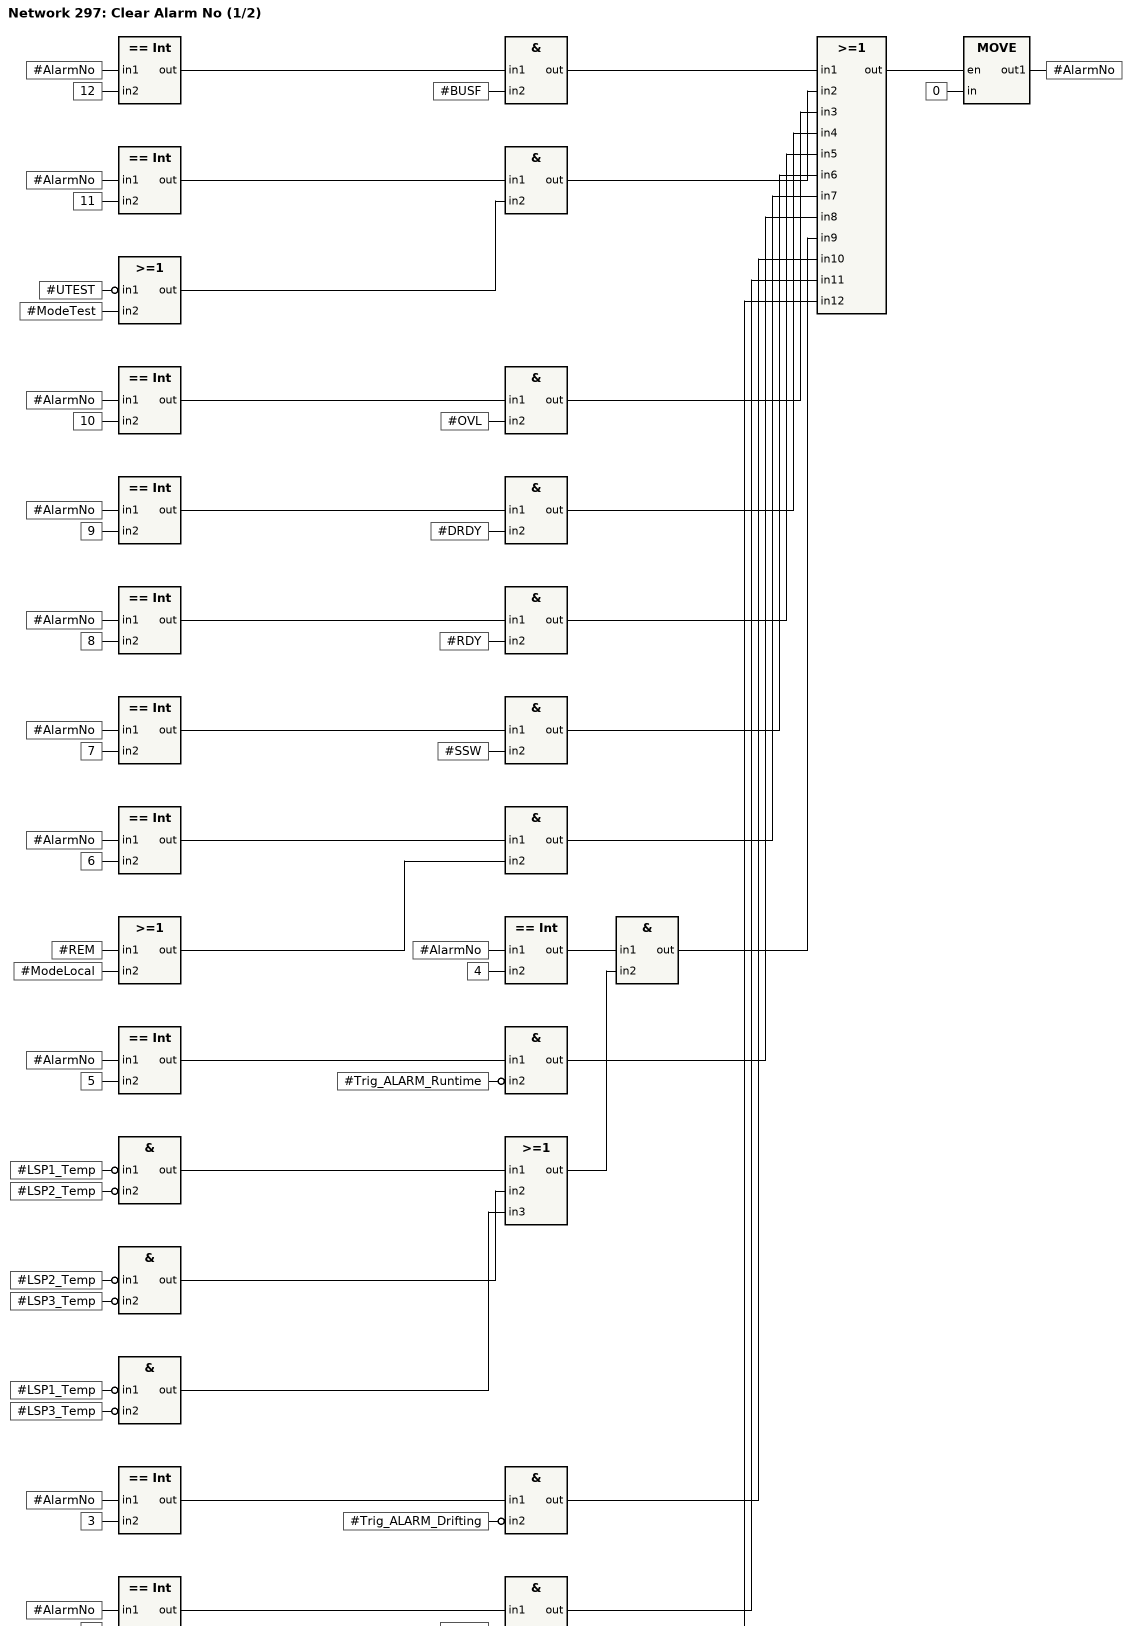
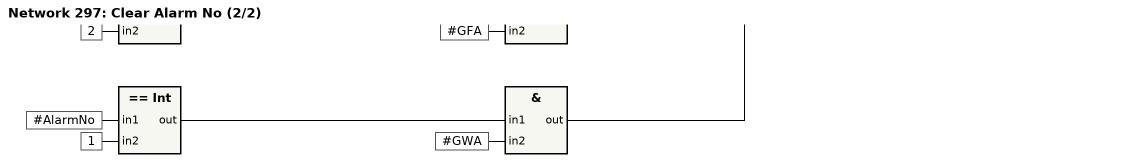
   IF ((#AlarmNo = 12) AND #BUSF) OR ((#AlarmNo = 11) AND (NOT #UTEST OR #ModeTest)) OR ((#AlarmNo = 10) AND #OVL) OR ((#AlarmNo = 9) AND #DRDY) OR ((#AlarmNo = 8) AND #RDY) OR ((#AlarmNo = 7) AND #SSW) OR ((#AlarmNo = 6) AND (#REM OR #ModeLocal)) OR ((#AlarmNo = 5) AND NOT #Trig_ALARM_Runtime) OR ((#AlarmNo = 4) AND ((NOT #LSP1_Temp AND NOT #LSP2_Temp) OR (NOT #LSP2_Temp AND NOT #LSP3_Temp) OR (NOT #LSP1_Temp AND NOT #LSP3_Temp))) OR ((#AlarmNo = 3) AND NOT #Trig_ALARM_Drifting) OR ((#AlarmNo = 2) AND #GFA) OR ((#AlarmNo = 1) AND #GWA) THEN
       #AlarmNo := 0;
   END_IF;
END_REGION

REGION Network 298: Clear Alarm No Old
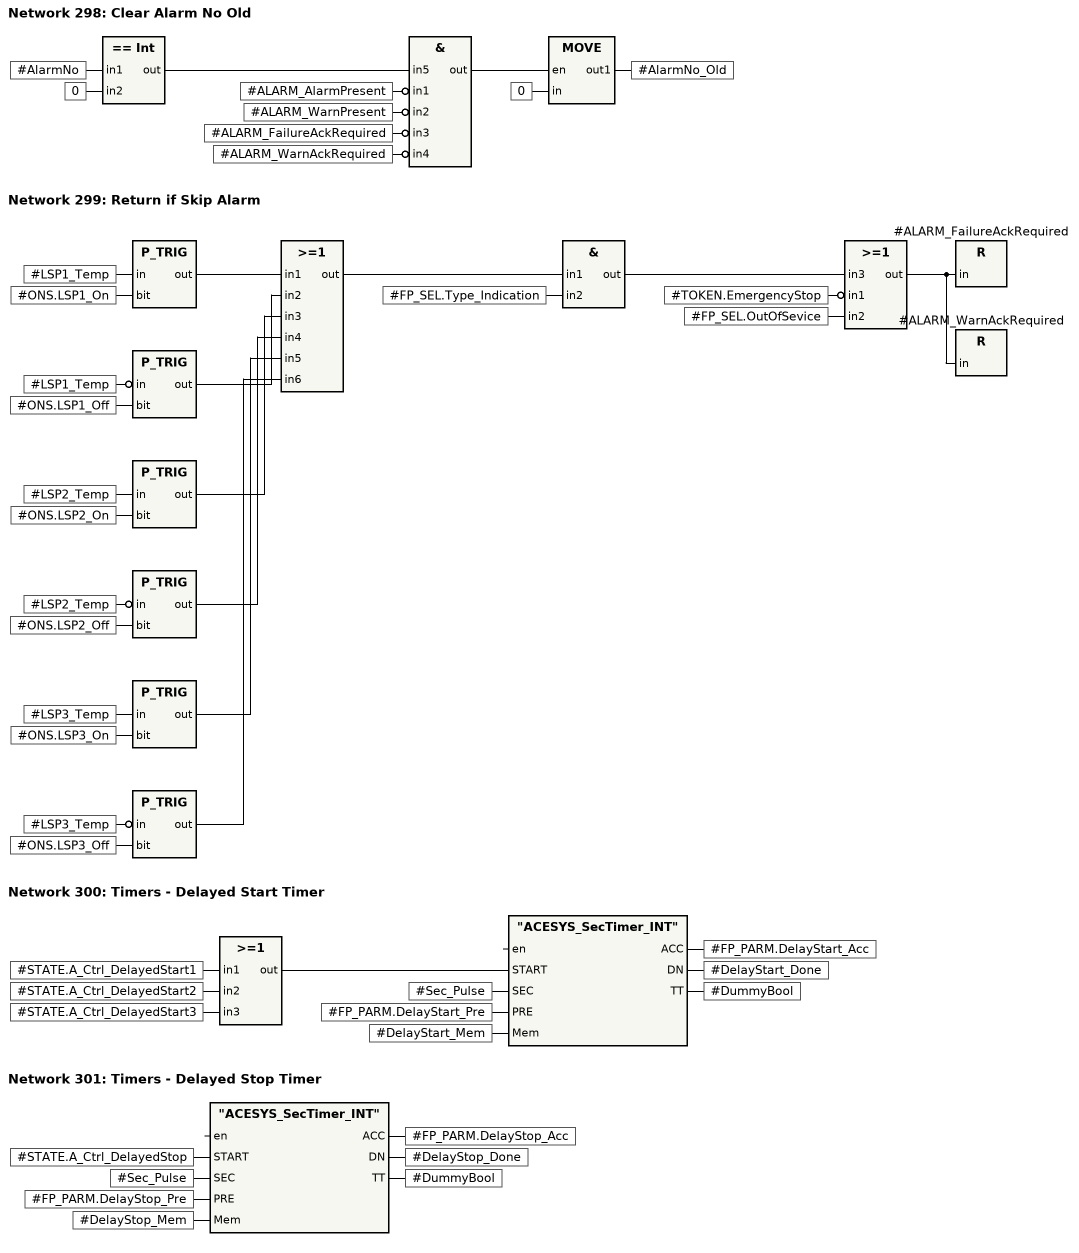
   IF (#AlarmNo = 0) AND NOT #ALARM_AlarmPresent AND NOT #ALARM_WarnPresent AND NOT #ALARM_FailureAckRequired AND NOT #ALARM_WarnAckRequired THEN
       #AlarmNo_Old := 0;
   END_IF;
END_REGION

REGION Network 299: Return if Skip Alarm
   // Build 002 - 27 March 2019 : Alarm/Warning are Auto Acknowledged on OutOfService
   // Build 003 - 30 June 2019 : Acknowledge pending alarms when Unit started as "Indication"
   Skip:
   #_w1 := #LSP1_Temp AND NOT #ONS.LSP1_On;   // rising edge
   #ONS.LSP1_On := #LSP1_Temp;
   #_w2 := NOT #LSP1_Temp AND NOT #ONS.LSP1_Off;   // rising edge
   #ONS.LSP1_Off := NOT #LSP1_Temp;
   #_w3 := #LSP2_Temp AND NOT #ONS.LSP2_On;   // rising edge
   #ONS.LSP2_On := #LSP2_Temp;
   #_w4 := NOT #LSP2_Temp AND NOT #ONS.LSP2_Off;   // rising edge
   #ONS.LSP2_Off := NOT #LSP2_Temp;
   #_w5 := #LSP3_Temp AND NOT #ONS.LSP3_On;   // rising edge
   #ONS.LSP3_On := #LSP3_Temp;
   #_w6 := NOT #LSP3_Temp AND NOT #ONS.LSP3_Off;   // rising edge
   #ONS.LSP3_Off := NOT #LSP3_Temp;
   IF ((#_w1 OR #_w2 OR #_w3 OR #_w4 OR #_w5 OR #_w6) AND #FP_SEL.Type_Indication) OR NOT #TOKEN.EmergencyStop OR #FP_SEL.OutOfSevice THEN
       #ALARM_FailureAckRequired := FALSE;
       #ALARM_WarnAckRequired := FALSE;
   END_IF;
END_REGION

REGION Network 300: Timers - Delayed Start Timer
   "ACESYS_SecTimer_INT"(START := #STATE.A_Ctrl_DelayedStart1 OR #STATE.A_Ctrl_DelayedStart2 OR #STATE.A_Ctrl_DelayedStart3,
                         SEC := #Sec_Pulse,
                         PRE := #FP_PARM.DelayStart_Pre,
                         Mem := #DelayStart_Mem,
                         ACC => #FP_PARM.DelayStart_Acc,
                         DN => #DelayStart_Done,
                         TT => #DummyBool);
END_REGION

REGION Network 301: Timers - Delayed Stop Timer
   "ACESYS_SecTimer_INT"(START := #STATE.A_Ctrl_DelayedStop,
                         SEC := #Sec_Pulse,
                         PRE := #FP_PARM.DelayStop_Pre,
                         Mem := #DelayStop_Mem,
                         ACC => #FP_PARM.DelayStop_Acc,
                         DN => #DelayStop_Done,
                         TT => #DummyBool);
END_REGION

REGION Network 302: Timers - Start Warning Timer
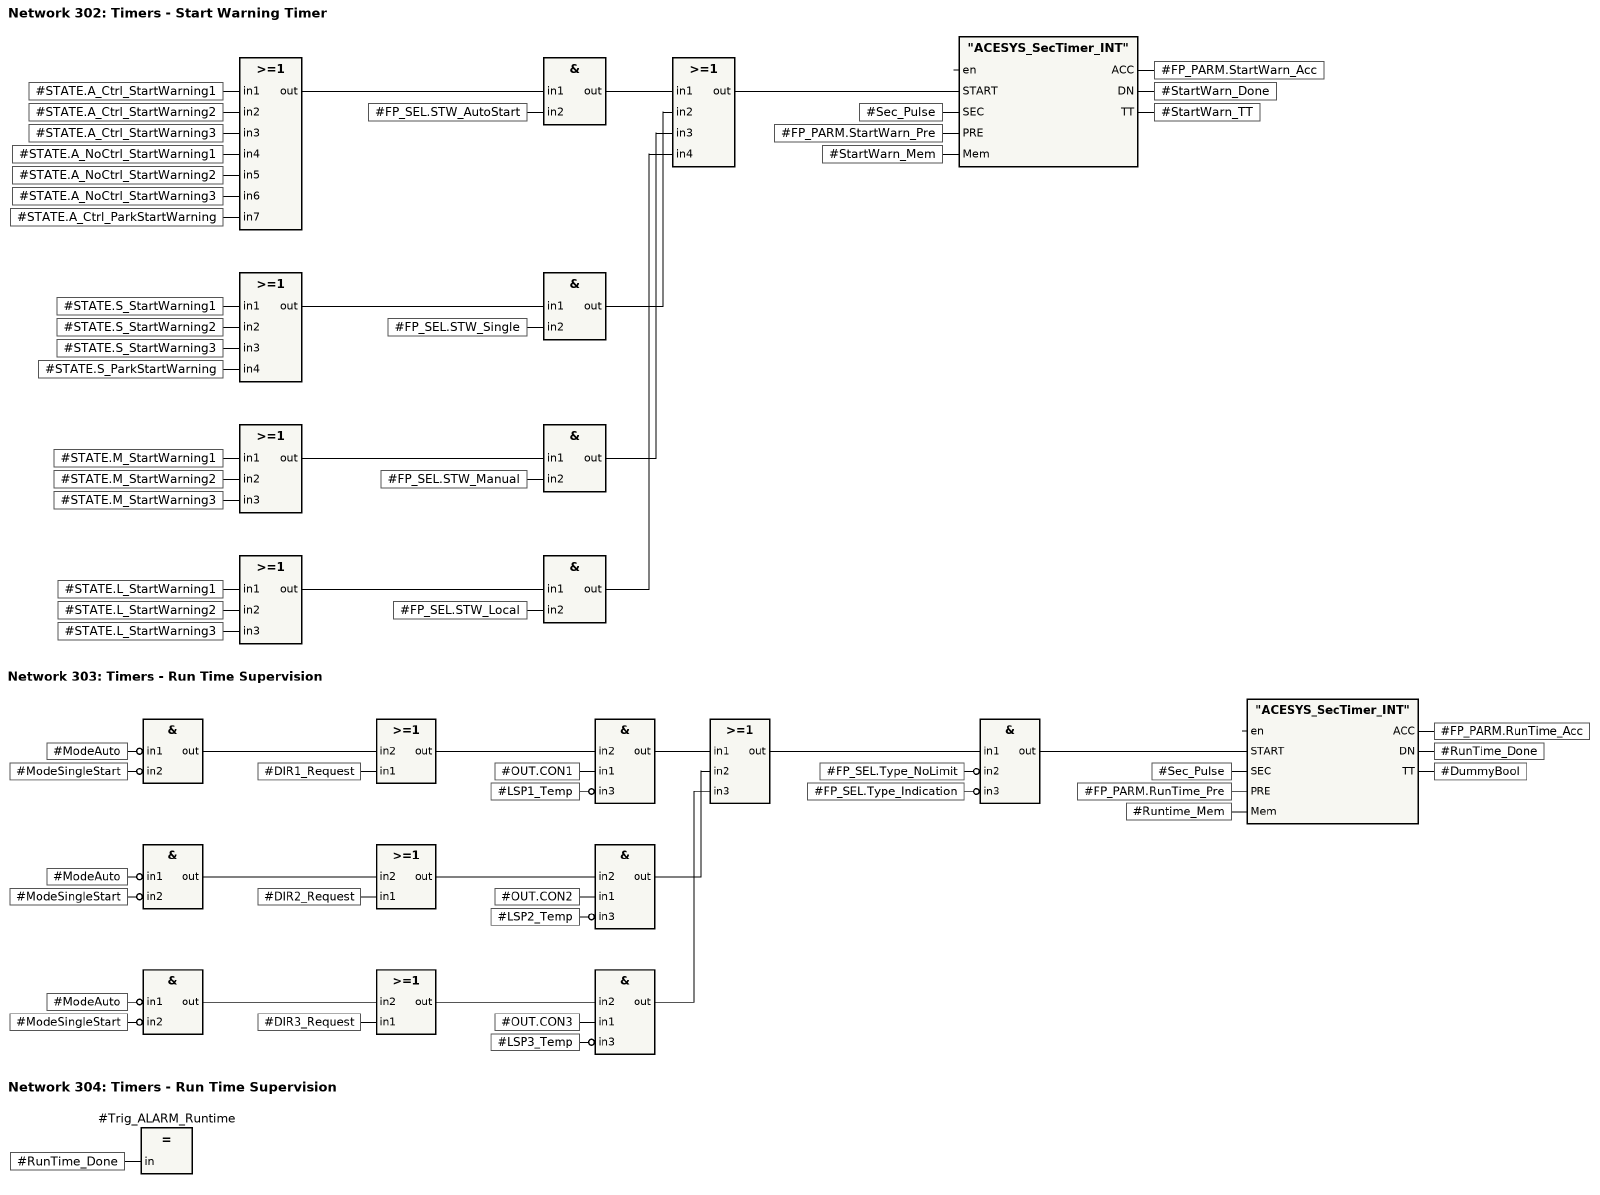
   "ACESYS_SecTimer_INT"(START := ((#STATE.A_Ctrl_StartWarning1 OR #STATE.A_Ctrl_StartWarning2 OR #STATE.A_Ctrl_StartWarning3 OR #STATE.A_NoCtrl_StartWarning1 OR #STATE.A_NoCtrl_StartWarning2 OR #STATE.A_NoCtrl_StartWarning3 OR #STATE.A_Ctrl_ParkStartWarning) AND #FP_SEL.STW_AutoStart) OR ((#STATE.S_StartWarning1 OR #STATE.S_StartWarning2 OR #STATE.S_StartWarning3 OR #STATE.S_ParkStartWarning) AND #FP_SEL.STW_Single) OR ((#STATE.M_StartWarning1 OR #STATE.M_StartWarning2 OR #STATE.M_StartWarning3) AND #FP_SEL.STW_Manual) OR ((#STATE.L_StartWarning1 OR #STATE.L_StartWarning2 OR #STATE.L_StartWarning3) AND #FP_SEL.STW_Local),
                         SEC := #Sec_Pulse,
                         PRE := #FP_PARM.StartWarn_Pre,
                         Mem := #StartWarn_Mem,
                         ACC => #FP_PARM.StartWarn_Acc,
                         DN => #StartWarn_Done,
                         TT => #StartWarn_TT);
END_REGION

REGION Network 303: Timers - Run Time Supervision
   "ACESYS_SecTimer_INT"(START := ((((NOT #ModeAuto AND NOT #ModeSingleStart) OR #DIR1_Request) AND #OUT.CON1 AND NOT #LSP1_Temp) OR (((NOT #ModeAuto AND NOT #ModeSingleStart) OR #DIR2_Request) AND #OUT.CON2 AND NOT #LSP2_Temp) OR (((NOT #ModeAuto AND NOT #ModeSingleStart) OR #DIR3_Request) AND #OUT.CON3 AND NOT #LSP3_Temp)) AND NOT #FP_SEL.Type_NoLimit AND NOT #FP_SEL.Type_Indication,
                         SEC := #Sec_Pulse,
                         PRE := #FP_PARM.RunTime_Pre,
                         Mem := #Runtime_Mem,
                         ACC => #FP_PARM.RunTime_Acc,
                         DN => #RunTime_Done,
                         TT => #DummyBool);
END_REGION

REGION Network 304: Timers - Run Time Supervision
   #Trig_ALARM_Runtime := #RunTime_Done;
END_REGION

REGION Network 305: Outputs - CON1
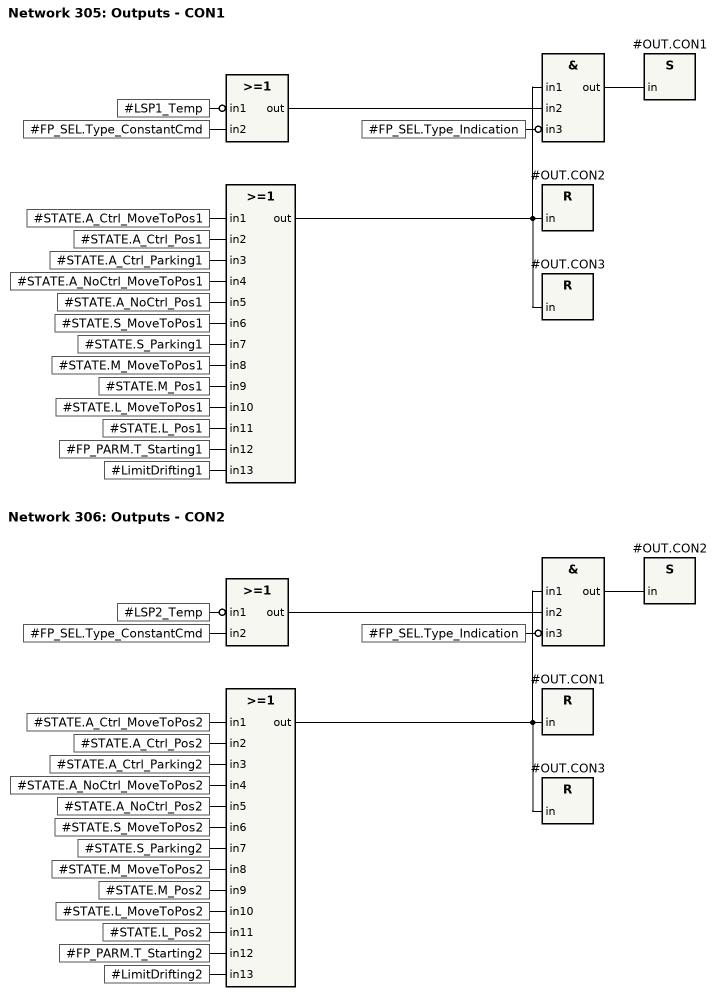
   #_w1 := #STATE.A_Ctrl_MoveToPos1 OR #STATE.A_Ctrl_Pos1 OR #STATE.A_Ctrl_Parking1 OR #STATE.A_NoCtrl_MoveToPos1 OR #STATE.A_NoCtrl_Pos1 OR #STATE.S_MoveToPos1 OR #STATE.S_Parking1 OR #STATE.M_MoveToPos1 OR #STATE.M_Pos1 OR #STATE.L_MoveToPos1 OR #STATE.L_Pos1 OR #FP_PARM.T_Starting1 OR #LimitDrifting1;
   IF #_w1 AND (NOT #LSP1_Temp OR #FP_SEL.Type_ConstantCmd) AND NOT #FP_SEL.Type_Indication THEN
       #OUT.CON1 := TRUE;
   END_IF;
   IF #_w1 THEN
       #OUT.CON2 := FALSE;
       #OUT.CON3 := FALSE;
   END_IF;
END_REGION

REGION Network 306: Outputs - CON2
   #_w1 := #STATE.A_Ctrl_MoveToPos2 OR #STATE.A_Ctrl_Pos2 OR #STATE.A_Ctrl_Parking2 OR #STATE.A_NoCtrl_MoveToPos2 OR #STATE.A_NoCtrl_Pos2 OR #STATE.S_MoveToPos2 OR #STATE.S_Parking2 OR #STATE.M_MoveToPos2 OR #STATE.M_Pos2 OR #STATE.L_MoveToPos2 OR #STATE.L_Pos2 OR #FP_PARM.T_Starting2 OR #LimitDrifting2;
   IF #_w1 AND (NOT #LSP2_Temp OR #FP_SEL.Type_ConstantCmd) AND NOT #FP_SEL.Type_Indication THEN
       #OUT.CON2 := TRUE;
   END_IF;
   IF #_w1 THEN
       #OUT.CON1 := FALSE;
       #OUT.CON3 := FALSE;
   END_IF;
END_REGION

REGION Network 307: Outputs - CON3
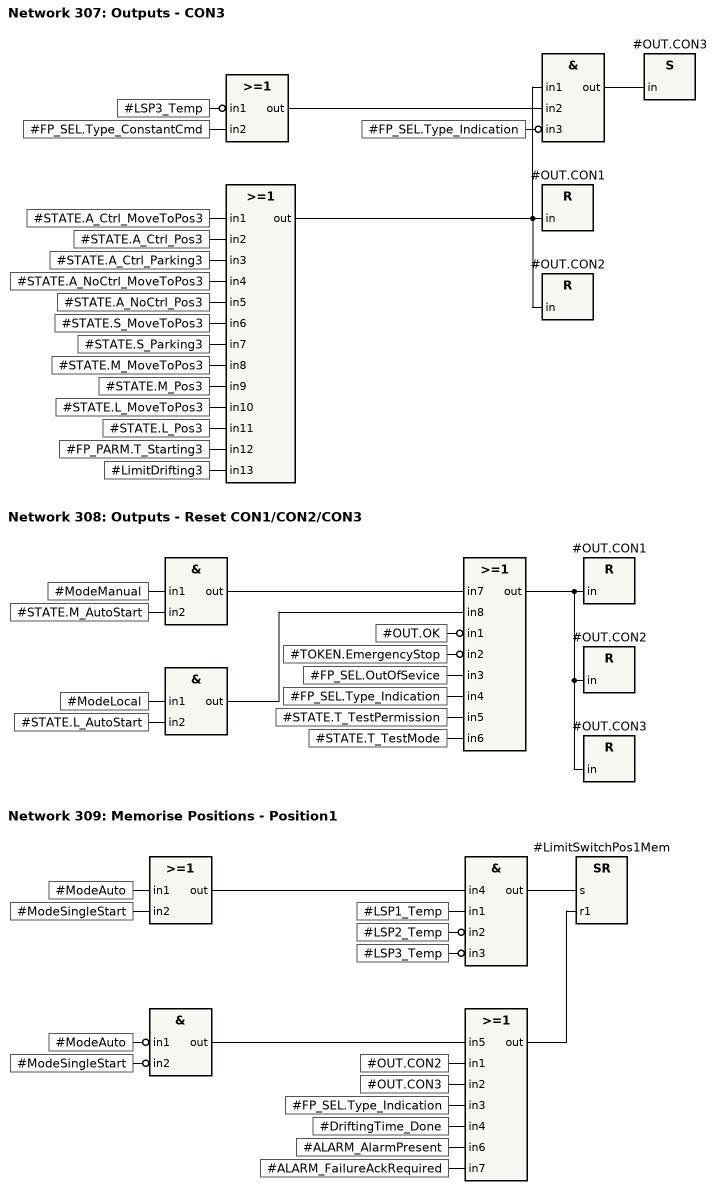
   #_w1 := #STATE.A_Ctrl_MoveToPos3 OR #STATE.A_Ctrl_Pos3 OR #STATE.A_Ctrl_Parking3 OR #STATE.A_NoCtrl_MoveToPos3 OR #STATE.A_NoCtrl_Pos3 OR #STATE.S_MoveToPos3 OR #STATE.S_Parking3 OR #STATE.M_MoveToPos3 OR #STATE.M_Pos3 OR #STATE.L_MoveToPos3 OR #STATE.L_Pos3 OR #FP_PARM.T_Starting3 OR #LimitDrifting3;
   IF #_w1 AND (NOT #LSP3_Temp OR #FP_SEL.Type_ConstantCmd) AND NOT #FP_SEL.Type_Indication THEN
       #OUT.CON3 := TRUE;
   END_IF;
   IF #_w1 THEN
       #OUT.CON1 := FALSE;
       #OUT.CON2 := FALSE;
   END_IF;
END_REGION

REGION Network 308: Outputs - Reset CON1/CON2/CON3
   // Build 002 - 27 March 2019 : Added TOKEN.EmergencyStop
   IF (#ModeManual AND #STATE.M_AutoStart) OR (#ModeLocal AND #STATE.L_AutoStart) OR NOT #OUT.OK OR NOT #TOKEN.EmergencyStop OR #FP_SEL.OutOfSevice OR #FP_SEL.Type_Indication OR #STATE.T_TestPermission OR #STATE.T_TestMode THEN
       #OUT.CON1 := FALSE;
       #OUT.CON2 := FALSE;
       #OUT.CON3 := FALSE;
   END_IF;
END_REGION

REGION Network 309: Memorise Positions - Position1
   // Build 002 - 27 March 2019 : Drfiting & memorise code are moved after CON code.
   // Build 005 - 11. Feb. 2020 : AlarmPresent & AlamAckRequired flag added to prevent drifiting during alarm
   IF (#ModeAuto OR #ModeSingleStart) AND #LSP1_Temp AND NOT #LSP2_Temp AND NOT #LSP3_Temp THEN
       #LimitSwitchPos1Mem := TRUE;   // SR flip-flop
   END_IF;
   IF (NOT #ModeAuto AND NOT #ModeSingleStart) OR #OUT.CON2 OR #OUT.CON3 OR #FP_SEL.Type_Indication OR #DriftingTime_Done OR #ALARM_AlarmPresent OR #ALARM_FailureAckRequired THEN
       #LimitSwitchPos1Mem := FALSE;
   END_IF;
END_REGION

REGION Network 310: Memorise Positions - Position2
   // Build 002 - 27 March 2019 : Drfiting & memorise code are moved after CON code.
   // Build 005 - 11. Feb. 2020 : AlarmPresent & AlamAckRequired flag added to prevent drifiting during alarm
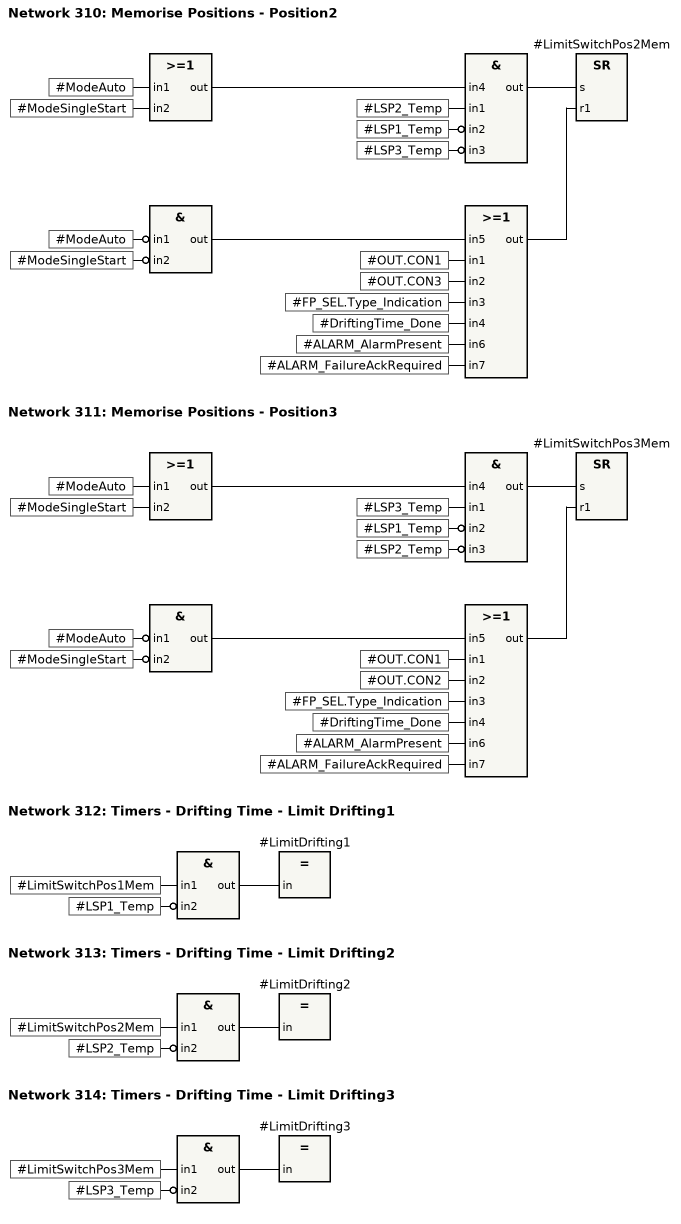
   IF (#ModeAuto OR #ModeSingleStart) AND #LSP2_Temp AND NOT #LSP1_Temp AND NOT #LSP3_Temp THEN
       #LimitSwitchPos2Mem := TRUE;   // SR flip-flop
   END_IF;
   IF (NOT #ModeAuto AND NOT #ModeSingleStart) OR #OUT.CON1 OR #OUT.CON3 OR #FP_SEL.Type_Indication OR #DriftingTime_Done OR #ALARM_AlarmPresent OR #ALARM_FailureAckRequired THEN
       #LimitSwitchPos2Mem := FALSE;
   END_IF;
END_REGION

REGION Network 311: Memorise Positions - Position3
   // Build 002 - 27 March 2019 : Drfiting & memorise code are moved after CON code.
   // Build 005 - 11. Feb. 2020 : AlarmPresent & AlamAckRequired flag added to prevent drifiting during alarm
   IF (#ModeAuto OR #ModeSingleStart) AND #LSP3_Temp AND NOT #LSP1_Temp AND NOT #LSP2_Temp THEN
       #LimitSwitchPos3Mem := TRUE;   // SR flip-flop
   END_IF;
   IF (NOT #ModeAuto AND NOT #ModeSingleStart) OR #OUT.CON1 OR #OUT.CON2 OR #FP_SEL.Type_Indication OR #DriftingTime_Done OR #ALARM_AlarmPresent OR #ALARM_FailureAckRequired THEN
       #LimitSwitchPos3Mem := FALSE;
   END_IF;
END_REGION

REGION Network 312: Timers - Drifting Time - Limit Drifting1
   // Build 002 - 27 March 2019 : Drfiting & memorise code are moved after CON code.
   #LimitDrifting1 := #LimitSwitchPos1Mem AND NOT #LSP1_Temp;
END_REGION

REGION Network 313: Timers - Drifting Time - Limit Drifting2
   // Build 002 - 27 March 2019 : Drfiting & memorise code are moved after CON code.
   #LimitDrifting2 := #LimitSwitchPos2Mem AND NOT #LSP2_Temp;
END_REGION

REGION Network 314: Timers - Drifting Time - Limit Drifting3
   // Build 002 - 27 March 2019 : Drfiting & memorise code are moved after CON code.
   #LimitDrifting3 := #LimitSwitchPos3Mem AND NOT #LSP3_Temp;
END_REGION

REGION Network 315: Timers - Drifting Time
   // Build 002 - 27 March 2019 : Drfiting & memorise code are moved after CON code.
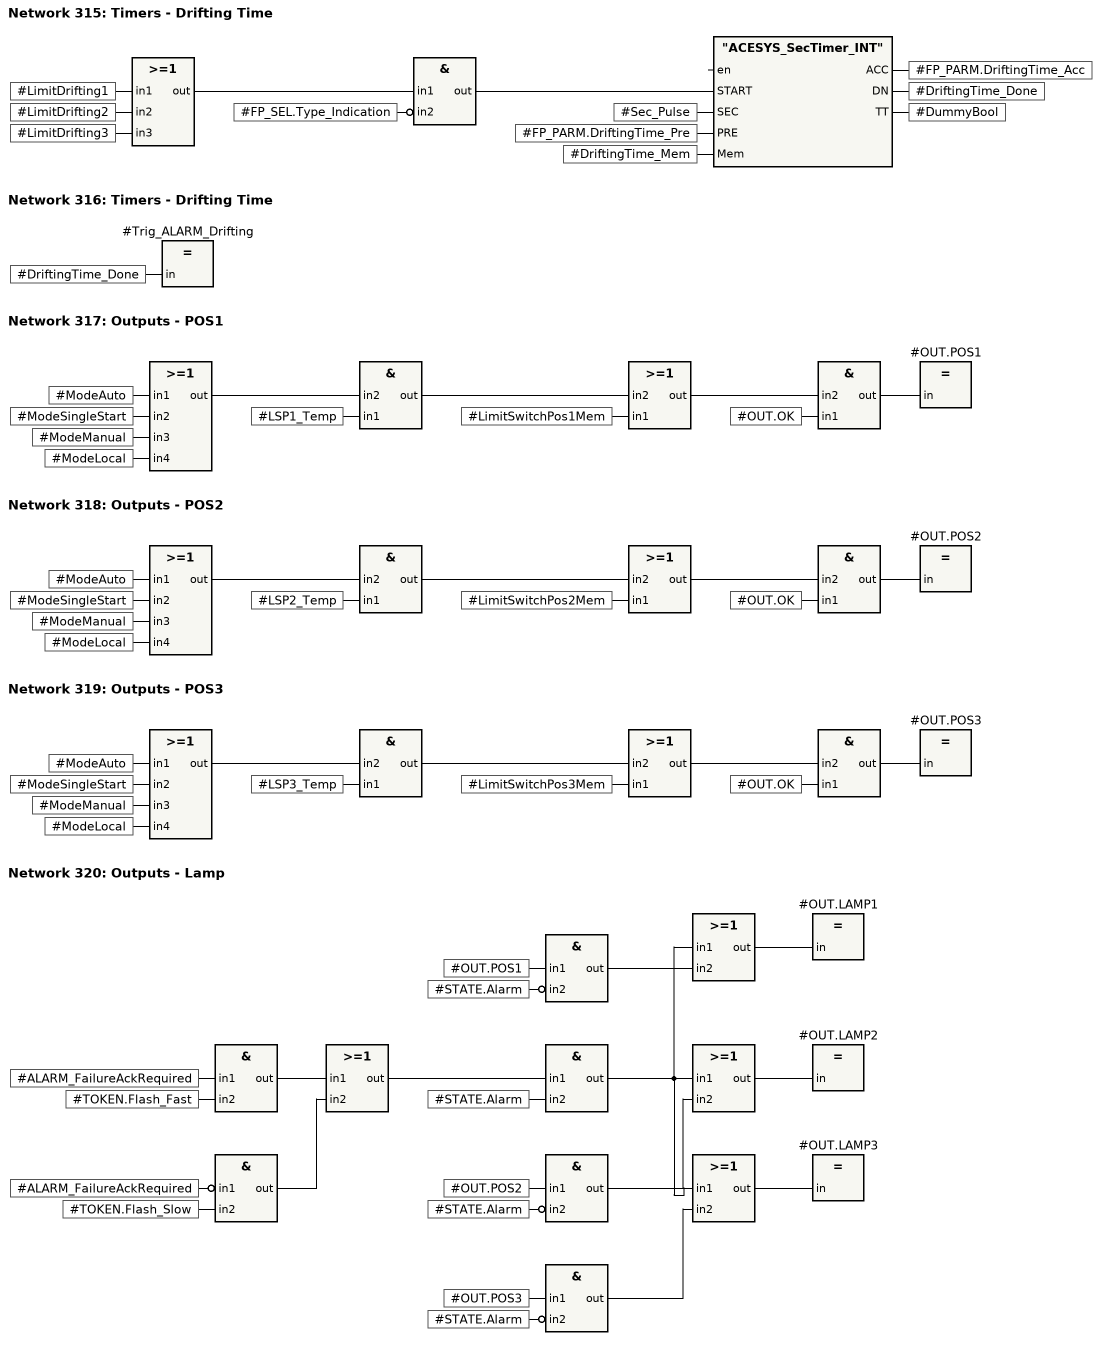
   "ACESYS_SecTimer_INT"(START := (#LimitDrifting1 OR #LimitDrifting2 OR #LimitDrifting3) AND NOT #FP_SEL.Type_Indication,
                         SEC := #Sec_Pulse,
                         PRE := #FP_PARM.DriftingTime_Pre,
                         Mem := #DriftingTime_Mem,
                         ACC => #FP_PARM.DriftingTime_Acc,
                         DN => #DriftingTime_Done,
                         TT => #DummyBool);
END_REGION

REGION Network 316: Timers - Drifting Time
   // Build 002 - 27 March 2019 : Drfiting & memorise code are moved after CON code.
   #Trig_ALARM_Drifting := #DriftingTime_Done;
END_REGION

REGION Network 317: Outputs - POS1
   #OUT.POS1 := (((#ModeAuto OR #ModeSingleStart OR #ModeManual OR #ModeLocal) AND #LSP1_Temp) OR #LimitSwitchPos1Mem) AND #OUT.OK;
END_REGION

REGION Network 318: Outputs - POS2
   #OUT.POS2 := (((#ModeAuto OR #ModeSingleStart OR #ModeManual OR #ModeLocal) AND #LSP2_Temp) OR #LimitSwitchPos2Mem) AND #OUT.OK;
END_REGION

REGION Network 319: Outputs - POS3
   #OUT.POS3 := (((#ModeAuto OR #ModeSingleStart OR #ModeManual OR #ModeLocal) AND #LSP3_Temp) OR #LimitSwitchPos3Mem) AND #OUT.OK;
END_REGION

REGION Network 320: Outputs - Lamp
   #_w1 := ((#ALARM_FailureAckRequired AND #TOKEN.Flash_Fast) OR (NOT #ALARM_FailureAckRequired AND #TOKEN.Flash_Slow)) AND #STATE.Alarm;
   #OUT.LAMP1 := #_w1 OR (#OUT.POS1 AND NOT #STATE.Alarm);
   #OUT.LAMP2 := #_w1 OR (#OUT.POS2 AND NOT #STATE.Alarm);
   #OUT.LAMP3 := #_w1 OR (#OUT.POS3 AND NOT #STATE.Alarm);
END_REGION

REGION Network 321: Outputs - Test Mode
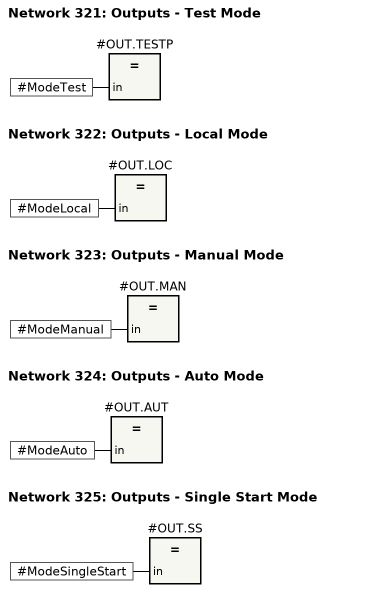
   #OUT.TESTP := #ModeTest;
END_REGION

REGION Network 322: Outputs - Local Mode
   #OUT.LOC := #ModeLocal;
END_REGION

REGION Network 323: Outputs - Manual Mode
   #OUT.MAN := #ModeManual;
END_REGION

REGION Network 324: Outputs - Auto Mode
   #OUT.AUT := #ModeAuto;
END_REGION

REGION Network 325: Outputs - Single Start Mode
   #OUT.SS := #ModeSingleStart;
END_REGION

REGION Network 326: Outputs - SACK
   // Build 003 - 08. Jul 2019 (EXTBOB) : FP_Sel.OutOfService flag  Deselect added on NonGroupCtrl Mode
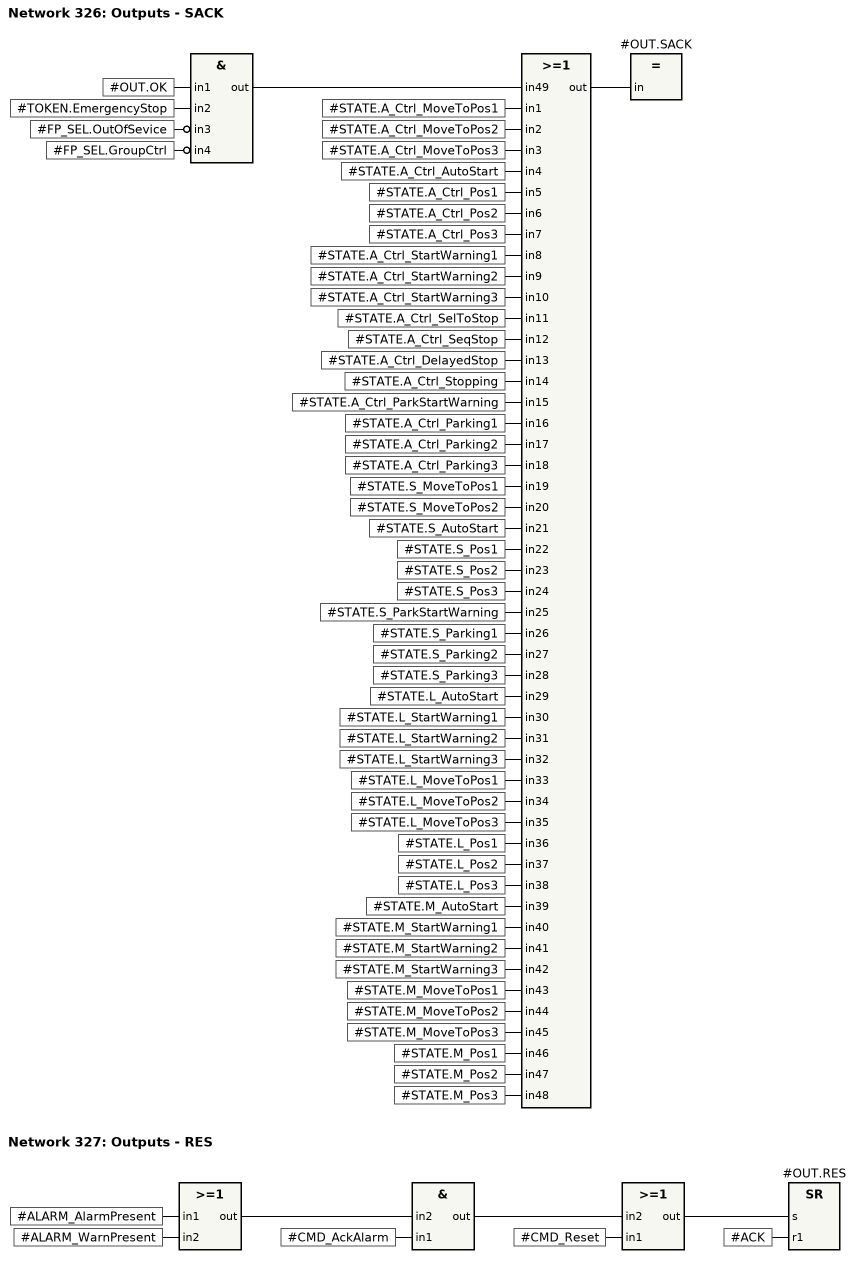
   #OUT.SACK := (#OUT.OK AND #TOKEN.EmergencyStop AND NOT #FP_SEL.OutOfSevice AND NOT #FP_SEL.GroupCtrl) OR #STATE.A_Ctrl_MoveToPos1 OR #STATE.A_Ctrl_MoveToPos2 OR #STATE.A_Ctrl_MoveToPos3 OR #STATE.A_Ctrl_AutoStart OR #STATE.A_Ctrl_Pos1 OR #STATE.A_Ctrl_Pos2 OR #STATE.A_Ctrl_Pos3 OR #STATE.A_Ctrl_StartWarning1 OR #STATE.A_Ctrl_StartWarning2 OR #STATE.A_Ctrl_StartWarning3 OR #STATE.A_Ctrl_SelToStop OR #STATE.A_Ctrl_SeqStop OR #STATE.A_Ctrl_DelayedStop OR #STATE.A_Ctrl_Stopping OR #STATE.A_Ctrl_ParkStartWarning OR #STATE.A_Ctrl_Parking1 OR #STATE.A_Ctrl_Parking2 OR #STATE.A_Ctrl_Parking3 OR #STATE.S_MoveToPos1 OR #STATE.S_MoveToPos2 OR #STATE.S_AutoStart OR #STATE.S_Pos1 OR #STATE.S_Pos2 OR #STATE.S_Pos3 OR #STATE.S_ParkStartWarning OR #STATE.S_Parking1 OR #STATE.S_Parking2 OR #STATE.S_Parking3 OR #STATE.L_AutoStart OR #STATE.L_StartWarning1 OR #STATE.L_StartWarning2 OR #STATE.L_StartWarning3 OR #STATE.L_MoveToPos1 OR #STATE.L_MoveToPos2 OR #STATE.L_MoveToPos3 OR #STATE.L_Pos1 OR #STATE.L_Pos2 OR #STATE.L_Pos3 OR #STATE.M_AutoStart OR #STATE.M_StartWarning1 OR #STATE.M_StartWarning2 OR #STATE.M_StartWarning3 OR #STATE.M_MoveToPos1 OR #STATE.M_MoveToPos2 OR #STATE.M_MoveToPos3 OR #STATE.M_Pos1 OR #STATE.M_Pos2 OR #STATE.M_Pos3;
END_REGION

REGION Network 327: Outputs - RES
   IF ((#ALARM_AlarmPresent OR #ALARM_WarnPresent) AND #CMD_AckAlarm) OR #CMD_Reset THEN
       #OUT.RES := TRUE;   // SR flip-flop
   END_IF;
   IF #ACK THEN #OUT.RES := FALSE; END_IF;
END_REGION

REGION Network 328: Outputs - OK
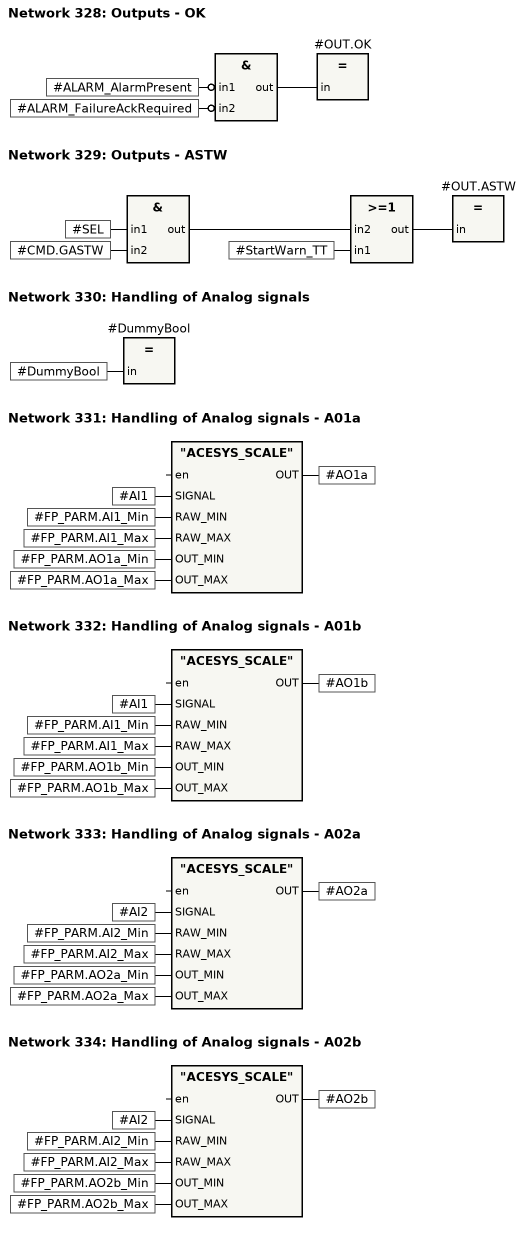
   #OUT.OK := NOT #ALARM_AlarmPresent AND NOT #ALARM_FailureAckRequired;
END_REGION

REGION Network 329: Outputs - ASTW
   #OUT.ASTW := (#SEL AND #CMD.GASTW) OR #StartWarn_TT;
END_REGION

REGION Network 330: Handling of Analog signals
   // ********************************************************************************
   // The block handles up to 3 analog signals.
   // 
   // The signals are AI1, AI2 and AI3 they are defined as reals.
   // 
   // By configuration at runtime these analog signals are converted into each 2 
   // values.
   // 
   // The parametres given from ECS defines:
   // 
   // 1) Min and Max for the input signal
   // 2) Corresponding Min and Max for Analog output "a"
   // 3) Corresponding Min and Max for Analog output "b"
   // 
   // Output a and b can be used for for instance a value in % and one in engineering 
   // units.
   // 
   // An example could be:
   // A motor current with a norminal value of 75 A
   // Input : motor current in mA; min=0, max = 75000
   // 
   // The signals are calculated by defining the formula for the line
   // 
   // Y = aX+b
   // 
   // Where a = (Y2 - Y1)/(X2-X1)
   // and   b = Y2 - aX2
   // Output a : motor current in %; min = 0, max = 100
   // output b : motor current in A; min = 0, max = 75
   #DummyBool := #DummyBool;
END_REGION

REGION Network 331: Handling of Analog signals - A01a
   "ACESYS_SCALE"(SIGNAL := #AI1,
                  RAW_MIN := #FP_PARM.AI1_Min,
                  RAW_MAX := #FP_PARM.AI1_Max,
                  OUT_MIN := #FP_PARM.AO1a_Min,
                  OUT_MAX := #FP_PARM.AO1a_Max,
                  OUT => #AO1a);
END_REGION

REGION Network 332: Handling of Analog signals - A01b
   "ACESYS_SCALE"(SIGNAL := #AI1,
                  RAW_MIN := #FP_PARM.AI1_Min,
                  RAW_MAX := #FP_PARM.AI1_Max,
                  OUT_MIN := #FP_PARM.AO1b_Min,
                  OUT_MAX := #FP_PARM.AO1b_Max,
                  OUT => #AO1b);
END_REGION

REGION Network 333: Handling of Analog signals - A02a
   "ACESYS_SCALE"(SIGNAL := #AI2,
                  RAW_MIN := #FP_PARM.AI2_Min,
                  RAW_MAX := #FP_PARM.AI2_Max,
                  OUT_MIN := #FP_PARM.AO2a_Min,
                  OUT_MAX := #FP_PARM.AO2a_Max,
                  OUT => #AO2a);
END_REGION

REGION Network 334: Handling of Analog signals - A02b
   "ACESYS_SCALE"(SIGNAL := #AI2,
                  RAW_MIN := #FP_PARM.AI2_Min,
                  RAW_MAX := #FP_PARM.AI2_Max,
                  OUT_MIN := #FP_PARM.AO2b_Min,
                  OUT_MAX := #FP_PARM.AO2b_Max,
                  OUT => #AO2b);
END_REGION

REGION Network 335: Handling of Analog signals - A03a
